  PROC DrawPart35()
    MoveL Offs(pOrigin,247.24,263.83,0.00),v40,z0,tPen\WObj:=wPaper;
    MoveL Offs(pOrigin,247.24,263.83,0.00),v40,z0,tPen\WObj:=wPaper;
    MoveL Offs(pOrigin,248.23,263.61,0.00),v40,z0,tPen\WObj:=wPaper;
    MoveL Offs(pOrigin,249.43,261.91,0.00),v40,z0,tPen\WObj:=wPaper;
    MoveL Offs(pOrigin,249.57,260.64,0.00),v40,z0,tPen\WObj:=wPaper;
    MoveL Offs(pOrigin,249.57,260.64,0.00),v40,z0,tPen\WObj:=wPaper;
    MoveL Offs(pOrigin,250.00,259.58,0.00),v40,z0,tPen\WObj:=wPaper;
    MoveL Offs(pOrigin,249.57,260.64,0.00),v40,z0,tPen\WObj:=wPaper;
    MoveL Offs(pOrigin,248.58,260.85,0.00),v40,z0,tPen\WObj:=wPaper;
    MoveL Offs(pOrigin,248.09,262.34,0.00),v40,z0,tPen\WObj:=wPaper;
    MoveL Offs(pOrigin,248.09,262.34,0.00),v40,z0,tPen\WObj:=wPaper;
    MoveL Offs(pOrigin,247.45,262.76,0.00),v40,z0,tPen\WObj:=wPaper;
    MoveL Offs(pOrigin,247.24,263.83,0.00),v40,fine,tPen\WObj:=wPaper;
    MoveL Offs(pOrigin,247.24,263.83,6.00),v60,z5,tPen\WObj:=wPaper;
    MoveL Offs(pOrigin,249.15,263.83,6.00),vTravel,z5,tPen\WObj:=wPaper;
    MoveL Offs(pOrigin,249.15,263.83,0.00),v60,z0,tPen\WObj:=wPaper;
    MoveL Offs(pOrigin,248.94,264.46,0.00),v40,z0,tPen\WObj:=wPaper;
    MoveL Offs(pOrigin,249.36,265.31,0.00),v40,z0,tPen\WObj:=wPaper;
    MoveL Offs(pOrigin,249.36,265.31,0.00),v40,z0,tPen\WObj:=wPaper;
    MoveL Offs(pOrigin,250.85,265.95,0.00),v40,z0,tPen\WObj:=wPaper;
    MoveL Offs(pOrigin,252.76,268.29,0.00),v40,z0,tPen\WObj:=wPaper;
    MoveL Offs(pOrigin,254.25,269.28,0.00),v40,z0,tPen\WObj:=wPaper;
    MoveL Offs(pOrigin,257.23,269.99,0.00),v40,z0,tPen\WObj:=wPaper;
    MoveL Offs(pOrigin,262.11,269.99,0.00),v40,z0,tPen\WObj:=wPaper;
    MoveL Offs(pOrigin,264.88,269.35,0.00),v40,z0,tPen\WObj:=wPaper;
    MoveL Offs(pOrigin,267.00,268.36,0.00),v40,z0,tPen\WObj:=wPaper;
    MoveL Offs(pOrigin,267.85,267.23,0.00),v40,z0,tPen\WObj:=wPaper;
    MoveL Offs(pOrigin,267.85,266.80,0.00),v40,z0,tPen\WObj:=wPaper;
    MoveL Offs(pOrigin,268.06,267.15,0.00),v40,z0,tPen\WObj:=wPaper;
    MoveL Offs(pOrigin,268.91,267.23,0.00),v40,z0,tPen\WObj:=wPaper;
    MoveL Offs(pOrigin,270.40,266.59,0.00),v40,fine,tPen\WObj:=wPaper;
    MoveL Offs(pOrigin,270.40,266.59,6.00),v60,z5,tPen\WObj:=wPaper;
    MoveL Offs(pOrigin,272.74,265.95,6.00),vTravel,z5,tPen\WObj:=wPaper;
    MoveL Offs(pOrigin,272.74,265.95,0.00),v60,z0,tPen\WObj:=wPaper;
    MoveL Offs(pOrigin,269.76,265.74,0.00),v40,z0,tPen\WObj:=wPaper;
    MoveL Offs(pOrigin,267.85,266.80,0.00),v40,z0,tPen\WObj:=wPaper;
    MoveL Offs(pOrigin,267.85,266.80,0.00),v40,z0,tPen\WObj:=wPaper;
    MoveL Offs(pOrigin,266.36,266.80,0.00),v40,z0,tPen\WObj:=wPaper;
    MoveL Offs(pOrigin,265.51,267.51,0.00),v40,z0,tPen\WObj:=wPaper;
    MoveL Offs(pOrigin,262.96,268.29,0.00),v40,z0,tPen\WObj:=wPaper;
    MoveL Offs(pOrigin,261.05,267.44,0.00),v40,z0,tPen\WObj:=wPaper;
    MoveL Offs(pOrigin,261.05,267.44,0.00),v40,z0,tPen\WObj:=wPaper;
    MoveL Offs(pOrigin,260.20,268.43,0.00),v40,z0,tPen\WObj:=wPaper;
    MoveL Offs(pOrigin,258.29,268.50,0.00),v40,z0,tPen\WObj:=wPaper;
    MoveL Offs(pOrigin,257.44,267.79,0.00),v40,z0,tPen\WObj:=wPaper;
    MoveL Offs(pOrigin,255.74,267.51,0.00),v40,z0,tPen\WObj:=wPaper;
    MoveL Offs(pOrigin,253.82,266.16,0.00),v40,z0,tPen\WObj:=wPaper;
    MoveL Offs(pOrigin,253.61,265.52,0.00),v40,z0,tPen\WObj:=wPaper;
    MoveL Offs(pOrigin,253.61,265.52,0.00),v40,z0,tPen\WObj:=wPaper;
    MoveL Offs(pOrigin,253.82,264.67,0.00),v40,z0,tPen\WObj:=wPaper;
    MoveL Offs(pOrigin,253.40,264.25,0.00),v40,z0,tPen\WObj:=wPaper;
    MoveL Offs(pOrigin,252.76,264.25,0.00),v40,z0,tPen\WObj:=wPaper;
    MoveL Offs(pOrigin,252.55,265.10,0.00),v40,z0,tPen\WObj:=wPaper;
    MoveL Offs(pOrigin,252.98,265.52,0.00),v40,z0,tPen\WObj:=wPaper;
    MoveL Offs(pOrigin,253.61,265.52,0.00),v40,z0,tPen\WObj:=wPaper;
    MoveL Offs(pOrigin,253.82,264.46,0.00),v40,z0,tPen\WObj:=wPaper;
    MoveL Offs(pOrigin,255.31,264.67,0.00),v40,z0,tPen\WObj:=wPaper;
    MoveL Offs(pOrigin,258.08,264.46,0.00),v40,z0,tPen\WObj:=wPaper;
    MoveL Offs(pOrigin,259.14,265.67,0.00),v40,z0,tPen\WObj:=wPaper;
    MoveL Offs(pOrigin,260.77,266.23,0.00),v40,z0,tPen\WObj:=wPaper;
    MoveL Offs(pOrigin,261.05,267.44,0.00),v40,fine,tPen\WObj:=wPaper;
    MoveL Offs(pOrigin,261.05,267.44,6.00),v60,z5,tPen\WObj:=wPaper;
    MoveL Offs(pOrigin,259.56,265.95,6.00),vTravel,z5,tPen\WObj:=wPaper;
    MoveL Offs(pOrigin,259.56,265.95,0.00),v60,z0,tPen\WObj:=wPaper;
    MoveL Offs(pOrigin,257.44,267.51,0.00),v40,z0,tPen\WObj:=wPaper;
    MoveL Offs(pOrigin,257.23,266.80,0.00),v40,z0,tPen\WObj:=wPaper;
    MoveL Offs(pOrigin,257.51,266.02,0.00),v40,z0,tPen\WObj:=wPaper;
    MoveL Offs(pOrigin,258.92,265.74,0.00),v40,z0,tPen\WObj:=wPaper;
    MoveL Offs(pOrigin,258.71,265.31,0.00),v40,z0,tPen\WObj:=wPaper;
    MoveL Offs(pOrigin,258.92,265.74,0.00),v40,z0,tPen\WObj:=wPaper;
    MoveL Offs(pOrigin,258.71,265.31,0.00),v40,fine,tPen\WObj:=wPaper;
    MoveL Offs(pOrigin,258.71,265.31,6.00),v60,z5,tPen\WObj:=wPaper;
    MoveL Offs(pOrigin,257.65,261.27,6.00),vTravel,z5,tPen\WObj:=wPaper;
    MoveL Offs(pOrigin,257.65,261.27,0.00),v60,z0,tPen\WObj:=wPaper;
    MoveL Offs(pOrigin,254.04,262.12,0.00),v40,fine,tPen\WObj:=wPaper;
    MoveL Offs(pOrigin,254.04,262.12,6.00),v60,z5,tPen\WObj:=wPaper;
    MoveL Offs(pOrigin,253.40,260.85,6.00),vTravel,z5,tPen\WObj:=wPaper;
    MoveL Offs(pOrigin,253.40,260.85,0.00),v60,z0,tPen\WObj:=wPaper;
    MoveL Offs(pOrigin,253.82,260.64,0.00),v40,z0,tPen\WObj:=wPaper;
    MoveL Offs(pOrigin,253.40,260.85,0.00),v40,fine,tPen\WObj:=wPaper;
    MoveL Offs(pOrigin,253.40,260.85,6.00),v60,z5,tPen\WObj:=wPaper;
    MoveL Offs(pOrigin,254.68,260.21,6.00),vTravel,z5,tPen\WObj:=wPaper;
    MoveL Offs(pOrigin,254.68,260.21,0.00),v60,z0,tPen\WObj:=wPaper;
    MoveL Offs(pOrigin,255.10,260.00,0.00),v40,z0,tPen\WObj:=wPaper;
    MoveL Offs(pOrigin,254.68,260.21,0.00),v40,fine,tPen\WObj:=wPaper;
    MoveL Offs(pOrigin,254.68,260.21,6.00),v60,z5,tPen\WObj:=wPaper;
    MoveL Offs(pOrigin,251.91,261.49,6.00),vTravel,z5,tPen\WObj:=wPaper;
    MoveL Offs(pOrigin,251.91,261.49,0.00),v60,z0,tPen\WObj:=wPaper;
    MoveL Offs(pOrigin,255.31,259.72,0.00),v40,z0,tPen\WObj:=wPaper;
    MoveL Offs(pOrigin,259.99,258.51,0.00),v40,fine,tPen\WObj:=wPaper;
    MoveL Offs(pOrigin,259.99,258.51,6.00),v60,z5,tPen\WObj:=wPaper;
    MoveL Offs(pOrigin,263.39,265.10,6.00),vTravel,z5,tPen\WObj:=wPaper;
    MoveL Offs(pOrigin,263.39,265.10,0.00),v60,z0,tPen\WObj:=wPaper;
    MoveL Offs(pOrigin,264.88,265.81,0.00),v40,z0,tPen\WObj:=wPaper;
    MoveL Offs(pOrigin,265.94,266.80,0.00),v40,fine,tPen\WObj:=wPaper;
    MoveL Offs(pOrigin,265.94,266.80,6.00),v60,z5,tPen\WObj:=wPaper;
    MoveL Offs(pOrigin,252.55,265.10,6.00),vTravel,z5,tPen\WObj:=wPaper;
    MoveL Offs(pOrigin,252.55,265.10,0.00),v60,z0,tPen\WObj:=wPaper;
    MoveL Offs(pOrigin,252.55,265.31,0.00),v40,z0,tPen\WObj:=wPaper;
    MoveL Offs(pOrigin,251.70,264.25,0.00),v40,z0,tPen\WObj:=wPaper;
    MoveL Offs(pOrigin,251.27,264.25,0.00),v40,fine,tPen\WObj:=wPaper;
    MoveL Offs(pOrigin,251.27,264.25,6.00),v60,z5,tPen\WObj:=wPaper;
    MoveL Offs(pOrigin,249.15,264.46,6.00),vTravel,z5,tPen\WObj:=wPaper;
    MoveL Offs(pOrigin,249.15,264.46,0.00),v60,z0,tPen\WObj:=wPaper;
    MoveL Offs(pOrigin,249.36,264.89,0.00),v40,z0,tPen\WObj:=wPaper;
    MoveL Offs(pOrigin,249.15,264.46,0.00),v40,fine,tPen\WObj:=wPaper;
    MoveL Offs(pOrigin,249.15,264.46,6.00),v60,z5,tPen\WObj:=wPaper;
    MoveL Offs(pOrigin,249.15,265.74,6.00),vTravel,z5,tPen\WObj:=wPaper;
    MoveL Offs(pOrigin,249.15,265.74,0.00),v60,z0,tPen\WObj:=wPaper;
    MoveL Offs(pOrigin,250.43,266.59,0.00),v40,z0,tPen\WObj:=wPaper;
    MoveL Offs(pOrigin,251.06,266.59,0.00),v40,fine,tPen\WObj:=wPaper;
    MoveL Offs(pOrigin,251.06,266.59,6.00),v60,z5,tPen\WObj:=wPaper;
    MoveL Offs(pOrigin,249.15,265.74,6.00),vTravel,z5,tPen\WObj:=wPaper;
    MoveL Offs(pOrigin,249.15,265.74,0.00),v60,z0,tPen\WObj:=wPaper;
    MoveL Offs(pOrigin,248.73,265.95,0.00),v40,z0,tPen\WObj:=wPaper;
    MoveL Offs(pOrigin,248.73,266.59,0.00),v40,fine,tPen\WObj:=wPaper;
    MoveL Offs(pOrigin,248.73,266.59,6.00),v60,z5,tPen\WObj:=wPaper;
    MoveL Offs(pOrigin,246.60,270.41,6.00),vTravel,z5,tPen\WObj:=wPaper;
    MoveL Offs(pOrigin,246.60,270.41,0.00),v60,z0,tPen\WObj:=wPaper;
    MoveL Offs(pOrigin,247.02,270.84,0.00),v40,z0,tPen\WObj:=wPaper;
  ENDPROC

  PROC DrawPart36()
    MoveL Offs(pOrigin,246.60,270.41,0.00),v40,fine,tPen\WObj:=wPaper;
    MoveL Offs(pOrigin,246.60,270.41,6.00),v60,z5,tPen\WObj:=wPaper;
    MoveL Offs(pOrigin,245.54,269.77,6.00),vTravel,z5,tPen\WObj:=wPaper;
    MoveL Offs(pOrigin,245.54,269.77,0.00),v60,z0,tPen\WObj:=wPaper;
    MoveL Offs(pOrigin,244.69,270.41,0.00),v40,z0,tPen\WObj:=wPaper;
    MoveL Offs(pOrigin,243.34,272.33,0.00),v40,z0,tPen\WObj:=wPaper;
    MoveL Offs(pOrigin,242.35,276.58,0.00),v40,fine,tPen\WObj:=wPaper;
    MoveL Offs(pOrigin,242.35,276.58,6.00),v60,z5,tPen\WObj:=wPaper;
    MoveL Offs(pOrigin,247.24,273.17,6.00),vTravel,z5,tPen\WObj:=wPaper;
    MoveL Offs(pOrigin,247.24,273.17,0.00),v60,z0,tPen\WObj:=wPaper;
    MoveL Offs(pOrigin,247.45,273.60,0.00),v40,z0,tPen\WObj:=wPaper;
    MoveL Offs(pOrigin,247.24,273.17,0.00),v40,z0,tPen\WObj:=wPaper;
    MoveL Offs(pOrigin,247.02,272.54,0.00),v40,z0,tPen\WObj:=wPaper;
    MoveL Offs(pOrigin,247.38,273.81,0.00),v40,z0,tPen\WObj:=wPaper;
    MoveL Offs(pOrigin,248.30,275.09,0.00),v40,fine,tPen\WObj:=wPaper;
    MoveL Offs(pOrigin,248.30,275.09,6.00),v60,z5,tPen\WObj:=wPaper;
    MoveL Offs(pOrigin,249.36,261.70,6.00),vTravel,z5,tPen\WObj:=wPaper;
    MoveL Offs(pOrigin,249.36,261.70,0.00),v60,z0,tPen\WObj:=wPaper;
    MoveL Offs(pOrigin,249.15,262.12,0.00),v40,z0,tPen\WObj:=wPaper;
    MoveL Offs(pOrigin,249.36,261.70,0.00),v40,fine,tPen\WObj:=wPaper;
    MoveL Offs(pOrigin,249.36,261.70,6.00),v60,z5,tPen\WObj:=wPaper;
    MoveL Offs(pOrigin,248.30,261.06,6.00),vTravel,z5,tPen\WObj:=wPaper;
    MoveL Offs(pOrigin,248.30,261.06,0.00),v60,z0,tPen\WObj:=wPaper;
    MoveL Offs(pOrigin,248.09,261.49,0.00),v40,z0,tPen\WObj:=wPaper;
    MoveL Offs(pOrigin,248.30,261.06,0.00),v40,fine,tPen\WObj:=wPaper;
    MoveL Offs(pOrigin,248.30,261.06,6.00),v60,z5,tPen\WObj:=wPaper;
    MoveL Offs(pOrigin,247.24,259.79,6.00),vTravel,z5,tPen\WObj:=wPaper;
    MoveL Offs(pOrigin,247.24,259.79,0.00),v60,z0,tPen\WObj:=wPaper;
    MoveL Offs(pOrigin,247.02,260.21,0.00),v40,z0,tPen\WObj:=wPaper;
    MoveL Offs(pOrigin,247.24,259.79,0.00),v40,fine,tPen\WObj:=wPaper;
    MoveL Offs(pOrigin,247.24,259.79,6.00),v60,z5,tPen\WObj:=wPaper;
    MoveL Offs(pOrigin,204.74,265.52,6.00),vTravel,z5,tPen\WObj:=wPaper;
    MoveL Offs(pOrigin,204.74,265.52,0.00),v60,z0,tPen\WObj:=wPaper;
    MoveL Offs(pOrigin,203.89,265.31,0.00),v40,z0,tPen\WObj:=wPaper;
    MoveL Offs(pOrigin,203.25,265.95,0.00),v40,z0,tPen\WObj:=wPaper;
    MoveL Offs(pOrigin,203.25,265.95,0.00),v40,z0,tPen\WObj:=wPaper;
    MoveL Offs(pOrigin,202.19,267.23,0.00),v40,z0,tPen\WObj:=wPaper;
    MoveL Offs(pOrigin,202.19,267.23,0.00),v40,z0,tPen\WObj:=wPaper;
    MoveL Offs(pOrigin,202.40,268.29,0.00),v40,z0,tPen\WObj:=wPaper;
    MoveL Offs(pOrigin,202.19,268.71,0.00),v40,fine,tPen\WObj:=wPaper;
    MoveL Offs(pOrigin,202.19,268.71,6.00),v60,z5,tPen\WObj:=wPaper;
    MoveL Offs(pOrigin,202.19,267.23,6.00),vTravel,z5,tPen\WObj:=wPaper;
    MoveL Offs(pOrigin,202.19,267.23,0.00),v60,z0,tPen\WObj:=wPaper;
    MoveL Offs(pOrigin,201.34,266.80,0.00),v40,z0,tPen\WObj:=wPaper;
    MoveL Offs(pOrigin,200.91,266.02,0.00),v40,z0,tPen\WObj:=wPaper;
    MoveL Offs(pOrigin,203.25,265.95,0.00),v40,z0,tPen\WObj:=wPaper;
    MoveL Offs(pOrigin,203.68,265.31,0.00),v40,z0,tPen\WObj:=wPaper;
    MoveL Offs(pOrigin,202.82,263.83,0.00),v40,z0,tPen\WObj:=wPaper;
    MoveL Offs(pOrigin,202.82,263.83,0.00),v40,z0,tPen\WObj:=wPaper;
    MoveL Offs(pOrigin,203.11,261.27,0.00),v40,z0,tPen\WObj:=wPaper;
    MoveL Offs(pOrigin,204.10,260.21,0.00),v40,fine,tPen\WObj:=wPaper;
    MoveL Offs(pOrigin,204.10,260.21,6.00),v60,z5,tPen\WObj:=wPaper;
    MoveL Offs(pOrigin,202.82,263.83,6.00),vTravel,z5,tPen\WObj:=wPaper;
    MoveL Offs(pOrigin,202.82,263.83,0.00),v60,z0,tPen\WObj:=wPaper;
    MoveL Offs(pOrigin,200.27,264.46,0.00),v40,fine,tPen\WObj:=wPaper;
    MoveL Offs(pOrigin,200.27,264.46,6.00),v60,z5,tPen\WObj:=wPaper;
    MoveL Offs(pOrigin,199.85,267.65,6.00),vTravel,z5,tPen\WObj:=wPaper;
    MoveL Offs(pOrigin,199.85,267.65,0.00),v60,z0,tPen\WObj:=wPaper;
    MoveL Offs(pOrigin,199.43,267.86,0.00),v40,z0,tPen\WObj:=wPaper;
    MoveL Offs(pOrigin,199.43,268.50,0.00),v40,z0,tPen\WObj:=wPaper;
    MoveL Offs(pOrigin,199.43,268.50,0.00),v40,z0,tPen\WObj:=wPaper;
    MoveL Offs(pOrigin,200.84,270.20,0.00),v40,z0,tPen\WObj:=wPaper;
    MoveL Offs(pOrigin,200.49,271.26,0.00),v40,z0,tPen\WObj:=wPaper;
    MoveL Offs(pOrigin,200.49,271.26,0.00),v40,z0,tPen\WObj:=wPaper;
    MoveL Offs(pOrigin,201.55,274.45,0.00),v40,z0,tPen\WObj:=wPaper;
    MoveL Offs(pOrigin,201.34,275.09,0.00),v40,z0,tPen\WObj:=wPaper;
    MoveL Offs(pOrigin,201.34,275.09,0.00),v40,z0,tPen\WObj:=wPaper;
    MoveL Offs(pOrigin,202.90,278.27,0.00),v40,z0,tPen\WObj:=wPaper;
    MoveL Offs(pOrigin,203.25,279.76,0.00),v40,z0,tPen\WObj:=wPaper;
    MoveL Offs(pOrigin,203.25,279.76,0.00),v40,z0,tPen\WObj:=wPaper;
    MoveL Offs(pOrigin,204.17,280.61,0.00),v40,z0,tPen\WObj:=wPaper;
    MoveL Offs(pOrigin,204.95,282.74,0.00),v40,fine,tPen\WObj:=wPaper;
    MoveL Offs(pOrigin,204.95,282.74,6.00),v60,z5,tPen\WObj:=wPaper;
    MoveL Offs(pOrigin,204.95,284.44,6.00),vTravel,z5,tPen\WObj:=wPaper;
    MoveL Offs(pOrigin,204.95,284.44,0.00),v60,z0,tPen\WObj:=wPaper;
    MoveL Offs(pOrigin,204.31,283.66,0.00),v40,z0,tPen\WObj:=wPaper;
    MoveL Offs(pOrigin,203.46,283.66,0.00),v40,z0,tPen\WObj:=wPaper;
    MoveL Offs(pOrigin,203.25,285.08,0.00),v40,z0,tPen\WObj:=wPaper;
    MoveL Offs(pOrigin,203.25,285.08,0.00),v40,z0,tPen\WObj:=wPaper;
    MoveL Offs(pOrigin,204.45,285.71,0.00),v40,z0,tPen\WObj:=wPaper;
    MoveL Offs(pOrigin,206.23,289.54,0.00),v40,fine,tPen\WObj:=wPaper;
    MoveL Offs(pOrigin,206.23,289.54,6.00),v60,z5,tPen\WObj:=wPaper;
    MoveL Offs(pOrigin,204.95,290.17,6.00),vTravel,z5,tPen\WObj:=wPaper;
    MoveL Offs(pOrigin,204.95,290.17,0.00),v60,z0,tPen\WObj:=wPaper;
    MoveL Offs(pOrigin,205.45,290.39,0.00),v40,z0,tPen\WObj:=wPaper;
    MoveL Offs(pOrigin,206.86,292.73,0.00),v40,fine,tPen\WObj:=wPaper;
    MoveL Offs(pOrigin,206.86,292.73,6.00),v60,z5,tPen\WObj:=wPaper;
    MoveL Offs(pOrigin,204.52,291.02,6.00),vTravel,z5,tPen\WObj:=wPaper;
    MoveL Offs(pOrigin,204.52,291.02,0.00),v60,z0,tPen\WObj:=wPaper;
    MoveL Offs(pOrigin,204.74,291.45,0.00),v40,z0,tPen\WObj:=wPaper;
    MoveL Offs(pOrigin,204.52,291.02,0.00),v40,z0,tPen\WObj:=wPaper;
    MoveL Offs(pOrigin,204.52,290.39,0.00),v40,z0,tPen\WObj:=wPaper;
    MoveL Offs(pOrigin,204.31,290.81,0.00),v40,z0,tPen\WObj:=wPaper;
    MoveL Offs(pOrigin,204.74,291.66,0.00),v40,z0,tPen\WObj:=wPaper;
    MoveL Offs(pOrigin,208.14,295.70,0.00),v40,fine,tPen\WObj:=wPaper;
    MoveL Offs(pOrigin,208.14,295.70,6.00),v60,z5,tPen\WObj:=wPaper;
    MoveL Offs(pOrigin,205.80,296.55,6.00),vTravel,z5,tPen\WObj:=wPaper;
    MoveL Offs(pOrigin,205.80,296.55,0.00),v60,z0,tPen\WObj:=wPaper;
    MoveL Offs(pOrigin,204.95,294.85,0.00),v40,z0,tPen\WObj:=wPaper;
    MoveL Offs(pOrigin,201.48,290.81,0.00),v40,z0,tPen\WObj:=wPaper;
    MoveL Offs(pOrigin,198.57,285.50,0.00),v40,z0,tPen\WObj:=wPaper;
    MoveL Offs(pOrigin,198.57,285.50,0.00),v40,z0,tPen\WObj:=wPaper;
    MoveL Offs(pOrigin,198.50,284.44,0.00),v40,z0,tPen\WObj:=wPaper;
    MoveL Offs(pOrigin,196.95,282.52,0.00),v40,z0,tPen\WObj:=wPaper;
    MoveL Offs(pOrigin,196.66,281.67,0.00),v40,z0,tPen\WObj:=wPaper;
    MoveL Offs(pOrigin,196.88,281.11,0.00),v40,z0,tPen\WObj:=wPaper;
    MoveL Offs(pOrigin,197.30,281.04,0.00),v40,z0,tPen\WObj:=wPaper;
    MoveL Offs(pOrigin,197.30,281.04,0.00),v40,z0,tPen\WObj:=wPaper;
    MoveL Offs(pOrigin,198.57,281.89,0.00),v40,z0,tPen\WObj:=wPaper;
    MoveL Offs(pOrigin,201.98,286.35,0.00),v40,z0,tPen\WObj:=wPaper;
    MoveL Offs(pOrigin,201.98,286.35,0.00),v40,z0,tPen\WObj:=wPaper;
    MoveL Offs(pOrigin,203.11,287.84,0.00),v40,z0,tPen\WObj:=wPaper;
    MoveL Offs(pOrigin,203.68,289.75,0.00),v40,z0,tPen\WObj:=wPaper;
    MoveL Offs(pOrigin,203.68,289.75,0.00),v40,z0,tPen\WObj:=wPaper;
    MoveL Offs(pOrigin,203.04,290.60,0.00),v40,z0,tPen\WObj:=wPaper;
    MoveL Offs(pOrigin,203.25,291.88,0.00),v40,z0,tPen\WObj:=wPaper;
    MoveL Offs(pOrigin,203.04,292.30,0.00),v40,z0,tPen\WObj:=wPaper;
    MoveL Offs(pOrigin,203.46,292.94,0.00),v40,z0,tPen\WObj:=wPaper;
    MoveL Offs(pOrigin,203.89,293.36,0.00),v40,z0,tPen\WObj:=wPaper;
    MoveL Offs(pOrigin,203.46,292.94,0.00),v40,fine,tPen\WObj:=wPaper;
  ENDPROC

  PROC DrawPart37()
    MoveL Offs(pOrigin,203.46,292.94,6.00),v60,z5,tPen\WObj:=wPaper;
    MoveL Offs(pOrigin,200.49,292.94,6.00),vTravel,z5,tPen\WObj:=wPaper;
    MoveL Offs(pOrigin,200.49,292.94,0.00),v60,z0,tPen\WObj:=wPaper;
    MoveL Offs(pOrigin,203.46,296.76,0.00),v40,z0,tPen\WObj:=wPaper;
    MoveL Offs(pOrigin,203.46,296.76,0.00),v40,z0,tPen\WObj:=wPaper;
    MoveL Offs(pOrigin,205.59,297.19,0.00),v40,z0,tPen\WObj:=wPaper;
    MoveL Offs(pOrigin,205.59,297.19,0.00),v40,z0,tPen\WObj:=wPaper;
    MoveL Offs(pOrigin,206.44,298.89,0.00),v40,fine,tPen\WObj:=wPaper;
    MoveL Offs(pOrigin,206.44,298.89,6.00),v60,z5,tPen\WObj:=wPaper;
    MoveL Offs(pOrigin,206.01,300.16,6.00),vTravel,z5,tPen\WObj:=wPaper;
    MoveL Offs(pOrigin,206.01,300.16,0.00),v60,z0,tPen\WObj:=wPaper;
    MoveL Offs(pOrigin,205.80,299.95,0.00),v40,z0,tPen\WObj:=wPaper;
    MoveL Offs(pOrigin,205.59,300.16,0.00),v40,z0,tPen\WObj:=wPaper;
    MoveL Offs(pOrigin,206.01,300.38,0.00),v40,z0,tPen\WObj:=wPaper;
    MoveL Offs(pOrigin,206.01,300.38,0.00),v40,z0,tPen\WObj:=wPaper;
    MoveL Offs(pOrigin,206.23,301.44,0.00),v40,z0,tPen\WObj:=wPaper;
    MoveL Offs(pOrigin,206.23,301.44,0.00),v40,z0,tPen\WObj:=wPaper;
    MoveL Offs(pOrigin,207.29,301.86,0.00),v40,z0,tPen\WObj:=wPaper;
    MoveL Offs(pOrigin,207.29,301.86,0.00),v40,z0,tPen\WObj:=wPaper;
    MoveL Offs(pOrigin,207.71,304.62,0.00),v40,z0,tPen\WObj:=wPaper;
    MoveL Offs(pOrigin,207.71,304.62,0.00),v40,z0,tPen\WObj:=wPaper;
    MoveL Offs(pOrigin,206.01,304.48,0.00),v40,z0,tPen\WObj:=wPaper;
    MoveL Offs(pOrigin,205.16,305.05,0.00),v40,z0,tPen\WObj:=wPaper;
    MoveL Offs(pOrigin,204.10,305.05,0.00),v40,z0,tPen\WObj:=wPaper;
    MoveL Offs(pOrigin,201.55,304.27,0.00),v40,z0,tPen\WObj:=wPaper;
    MoveL Offs(pOrigin,197.94,302.22,0.00),v40,z0,tPen\WObj:=wPaper;
    MoveL Offs(pOrigin,196.88,301.23,0.00),v40,z0,tPen\WObj:=wPaper;
    MoveL Offs(pOrigin,195.32,298.89,0.00),v40,z0,tPen\WObj:=wPaper;
    MoveL Offs(pOrigin,194.25,295.91,0.00),v40,z0,tPen\WObj:=wPaper;
    MoveL Offs(pOrigin,193.26,295.06,0.00),v40,z0,tPen\WObj:=wPaper;
    MoveL Offs(pOrigin,193.26,295.06,0.00),v40,z0,tPen\WObj:=wPaper;
    MoveL Offs(pOrigin,192.77,292.30,0.00),v40,z0,tPen\WObj:=wPaper;
    MoveL Offs(pOrigin,193.90,291.45,0.00),v40,z0,tPen\WObj:=wPaper;
    MoveL Offs(pOrigin,193.90,291.45,0.00),v40,z0,tPen\WObj:=wPaper;
    MoveL Offs(pOrigin,192.62,290.60,0.00),v40,z0,tPen\WObj:=wPaper;
    MoveL Offs(pOrigin,192.41,291.02,0.00),v40,z0,tPen\WObj:=wPaper;
    MoveL Offs(pOrigin,192.41,291.02,0.00),v40,z0,tPen\WObj:=wPaper;
    MoveL Offs(pOrigin,192.62,292.09,0.00),v40,z0,tPen\WObj:=wPaper;
    MoveL Offs(pOrigin,192.41,291.02,0.00),v40,z0,tPen\WObj:=wPaper;
    MoveL Offs(pOrigin,191.35,291.52,0.00),v40,z0,tPen\WObj:=wPaper;
    MoveL Offs(pOrigin,190.85,292.51,0.00),v40,z0,tPen\WObj:=wPaper;
    MoveL Offs(pOrigin,189.86,295.91,0.00),v40,z0,tPen\WObj:=wPaper;
    MoveL Offs(pOrigin,189.65,298.04,0.00),v40,z0,tPen\WObj:=wPaper;
    MoveL Offs(pOrigin,190.43,301.23,0.00),v40,z0,tPen\WObj:=wPaper;
    MoveL Offs(pOrigin,192.70,305.48,0.00),v40,z0,tPen\WObj:=wPaper;
    MoveL Offs(pOrigin,193.48,307.60,0.00),v40,z0,tPen\WObj:=wPaper;
    MoveL Offs(pOrigin,193.48,307.60,0.00),v40,z0,tPen\WObj:=wPaper;
    MoveL Offs(pOrigin,194.75,307.95,0.00),v40,z0,tPen\WObj:=wPaper;
    MoveL Offs(pOrigin,195.81,309.09,0.00),v40,z0,tPen\WObj:=wPaper;
    MoveL Offs(pOrigin,195.81,309.09,0.00),v40,z0,tPen\WObj:=wPaper;
    MoveL Offs(pOrigin,196.45,310.15,0.00),v40,z0,tPen\WObj:=wPaper;
    MoveL Offs(pOrigin,199.00,311.50,0.00),v40,z0,tPen\WObj:=wPaper;
    MoveL Offs(pOrigin,201.12,312.06,0.00),v40,z0,tPen\WObj:=wPaper;
    MoveL Offs(pOrigin,203.46,312.06,0.00),v40,z0,tPen\WObj:=wPaper;
    MoveL Offs(pOrigin,207.71,310.43,0.00),v40,z0,tPen\WObj:=wPaper;
    MoveL Offs(pOrigin,209.62,309.09,0.00),v40,z0,tPen\WObj:=wPaper;
    MoveL Offs(pOrigin,210.26,308.02,0.00),v40,z0,tPen\WObj:=wPaper;
    MoveL Offs(pOrigin,210.26,308.02,0.00),v40,z0,tPen\WObj:=wPaper;
    MoveL Offs(pOrigin,212.39,307.60,0.00),v40,z0,tPen\WObj:=wPaper;
    MoveL Offs(pOrigin,214.73,307.81,0.00),v40,z0,tPen\WObj:=wPaper;
    MoveL Offs(pOrigin,218.34,307.60,0.00),v40,fine,tPen\WObj:=wPaper;
    MoveL Offs(pOrigin,218.34,307.60,6.00),v60,z5,tPen\WObj:=wPaper;
    MoveL Offs(pOrigin,215.79,306.33,6.00),vTravel,z5,tPen\WObj:=wPaper;
    MoveL Offs(pOrigin,215.79,306.33,0.00),v60,z0,tPen\WObj:=wPaper;
    MoveL Offs(pOrigin,210.69,306.11,0.00),v40,z0,tPen\WObj:=wPaper;
    MoveL Offs(pOrigin,209.77,306.96,0.00),v40,z0,tPen\WObj:=wPaper;
    MoveL Offs(pOrigin,210.26,308.02,0.00),v40,fine,tPen\WObj:=wPaper;
    MoveL Offs(pOrigin,210.26,308.02,6.00),v60,z5,tPen\WObj:=wPaper;
    MoveL Offs(pOrigin,207.93,307.39,6.00),vTravel,z5,tPen\WObj:=wPaper;
    MoveL Offs(pOrigin,207.93,307.39,0.00),v60,z0,tPen\WObj:=wPaper;
    MoveL Offs(pOrigin,207.93,307.81,0.00),v40,z0,tPen\WObj:=wPaper;
    MoveL Offs(pOrigin,206.86,308.66,0.00),v40,fine,tPen\WObj:=wPaper;
    MoveL Offs(pOrigin,206.86,308.66,6.00),v60,z5,tPen\WObj:=wPaper;
    MoveL Offs(pOrigin,203.89,308.02,6.00),vTravel,z5,tPen\WObj:=wPaper;
    MoveL Offs(pOrigin,203.89,308.02,0.00),v60,z0,tPen\WObj:=wPaper;
    MoveL Offs(pOrigin,203.89,306.96,0.00),v40,fine,tPen\WObj:=wPaper;
    MoveL Offs(pOrigin,203.89,306.96,6.00),v60,z5,tPen\WObj:=wPaper;
    MoveL Offs(pOrigin,200.91,305.90,6.00),vTravel,z5,tPen\WObj:=wPaper;
    MoveL Offs(pOrigin,200.91,305.90,0.00),v60,z0,tPen\WObj:=wPaper;
    MoveL Offs(pOrigin,204.31,306.96,0.00),v40,z0,tPen\WObj:=wPaper;
    MoveL Offs(pOrigin,207.29,306.96,0.00),v40,z0,tPen\WObj:=wPaper;
    MoveL Offs(pOrigin,208.35,307.39,0.00),v40,z0,tPen\WObj:=wPaper;
    MoveL Offs(pOrigin,209.20,307.32,0.00),v40,z0,tPen\WObj:=wPaper;
    MoveL Offs(pOrigin,209.34,306.75,0.00),v40,z0,tPen\WObj:=wPaper;
    MoveL Offs(pOrigin,208.14,304.62,0.00),v40,z0,tPen\WObj:=wPaper;
    MoveL Offs(pOrigin,208.14,304.62,0.00),v40,z0,tPen\WObj:=wPaper;
    MoveL Offs(pOrigin,209.41,304.20,0.00),v40,z0,tPen\WObj:=wPaper;
    MoveL Offs(pOrigin,214.73,305.05,0.00),v40,fine,tPen\WObj:=wPaper;
    MoveL Offs(pOrigin,214.73,305.05,6.00),v60,z5,tPen\WObj:=wPaper;
    MoveL Offs(pOrigin,213.45,303.56,6.00),vTravel,z5,tPen\WObj:=wPaper;
    MoveL Offs(pOrigin,213.45,303.56,0.00),v60,z0,tPen\WObj:=wPaper;
    MoveL Offs(pOrigin,207.71,301.65,0.00),v40,z0,tPen\WObj:=wPaper;
    MoveL Offs(pOrigin,207.29,301.86,0.00),v40,z0,tPen\WObj:=wPaper;
    MoveL Offs(pOrigin,206.23,301.44,0.00),v40,z0,tPen\WObj:=wPaper;
    MoveL Offs(pOrigin,205.59,301.86,0.00),v40,z0,tPen\WObj:=wPaper;
    MoveL Offs(pOrigin,203.68,301.51,0.00),v40,z0,tPen\WObj:=wPaper;
    MoveL Offs(pOrigin,199.21,298.89,0.00),v40,z0,tPen\WObj:=wPaper;
    MoveL Offs(pOrigin,197.30,296.98,0.00),v40,z0,tPen\WObj:=wPaper;
    MoveL Offs(pOrigin,193.90,291.45,0.00),v40,z0,tPen\WObj:=wPaper;
    MoveL Offs(pOrigin,193.69,291.02,0.00),v40,z0,tPen\WObj:=wPaper;
    MoveL Offs(pOrigin,193.90,291.45,0.00),v40,z0,tPen\WObj:=wPaper;
    MoveL Offs(pOrigin,193.69,291.02,0.00),v40,fine,tPen\WObj:=wPaper;
    MoveL Offs(pOrigin,193.69,291.02,6.00),v60,z5,tPen\WObj:=wPaper;
    MoveL Offs(pOrigin,192.41,290.60,6.00),vTravel,z5,tPen\WObj:=wPaper;
    MoveL Offs(pOrigin,192.41,290.60,0.00),v60,z0,tPen\WObj:=wPaper;
    MoveL Offs(pOrigin,191.77,288.48,0.00),v40,z0,tPen\WObj:=wPaper;
    MoveL Offs(pOrigin,191.77,286.35,0.00),v40,z0,tPen\WObj:=wPaper;
    MoveL Offs(pOrigin,191.77,286.35,0.00),v40,z0,tPen\WObj:=wPaper;
    MoveL Offs(pOrigin,191.56,284.44,0.00),v40,z0,tPen\WObj:=wPaper;
    MoveL Offs(pOrigin,191.77,282.52,0.00),v40,z0,tPen\WObj:=wPaper;
    MoveL Offs(pOrigin,192.20,281.67,0.00),v40,z0,tPen\WObj:=wPaper;
    MoveL Offs(pOrigin,193.05,281.25,0.00),v40,z0,tPen\WObj:=wPaper;
    MoveL Offs(pOrigin,193.05,281.25,0.00),v40,z0,tPen\WObj:=wPaper;
    MoveL Offs(pOrigin,193.69,281.89,0.00),v40,z0,tPen\WObj:=wPaper;
    MoveL Offs(pOrigin,194.32,283.59,0.00),v40,z0,tPen\WObj:=wPaper;
    MoveL Offs(pOrigin,194.32,283.59,0.00),v40,z0,tPen\WObj:=wPaper;
    MoveL Offs(pOrigin,195.60,283.87,0.00),v40,z0,tPen\WObj:=wPaper;
    MoveL Offs(pOrigin,198.57,285.50,0.00),v40,fine,tPen\WObj:=wPaper;
    MoveL Offs(pOrigin,198.57,285.50,6.00),v60,z5,tPen\WObj:=wPaper;
    MoveL Offs(pOrigin,199.85,287.41,6.00),vTravel,z5,tPen\WObj:=wPaper;
  ENDPROC

  PROC DrawPart38()
    MoveL Offs(pOrigin,199.85,287.41,0.00),v60,z0,tPen\WObj:=wPaper;
    MoveL Offs(pOrigin,200.06,287.84,0.00),v40,z0,tPen\WObj:=wPaper;
    MoveL Offs(pOrigin,199.85,287.41,0.00),v40,fine,tPen\WObj:=wPaper;
    MoveL Offs(pOrigin,199.85,287.41,6.00),v60,z5,tPen\WObj:=wPaper;
    MoveL Offs(pOrigin,201.98,286.35,6.00),vTravel,z5,tPen\WObj:=wPaper;
    MoveL Offs(pOrigin,201.98,286.35,0.00),v60,z0,tPen\WObj:=wPaper;
    MoveL Offs(pOrigin,202.61,285.71,0.00),v40,z0,tPen\WObj:=wPaper;
    MoveL Offs(pOrigin,203.04,285.71,0.00),v40,z0,tPen\WObj:=wPaper;
    MoveL Offs(pOrigin,203.04,285.71,0.00),v40,z0,tPen\WObj:=wPaper;
    MoveL Offs(pOrigin,203.25,286.56,0.00),v40,z0,tPen\WObj:=wPaper;
    MoveL Offs(pOrigin,202.82,286.99,0.00),v40,z0,tPen\WObj:=wPaper;
    MoveL Offs(pOrigin,203.04,287.41,0.00),v40,z0,tPen\WObj:=wPaper;
    MoveL Offs(pOrigin,203.25,287.84,0.00),v40,z0,tPen\WObj:=wPaper;
    MoveL Offs(pOrigin,203.04,287.41,0.00),v40,fine,tPen\WObj:=wPaper;
    MoveL Offs(pOrigin,203.04,287.41,6.00),v60,z5,tPen\WObj:=wPaper;
    MoveL Offs(pOrigin,202.19,285.92,6.00),vTravel,z5,tPen\WObj:=wPaper;
    MoveL Offs(pOrigin,202.19,285.92,0.00),v60,z0,tPen\WObj:=wPaper;
    MoveL Offs(pOrigin,201.98,286.35,0.00),v40,z0,tPen\WObj:=wPaper;
    MoveL Offs(pOrigin,202.19,285.92,0.00),v40,fine,tPen\WObj:=wPaper;
    MoveL Offs(pOrigin,202.19,285.92,6.00),v60,z5,tPen\WObj:=wPaper;
    MoveL Offs(pOrigin,203.25,283.59,6.00),vTravel,z5,tPen\WObj:=wPaper;
    MoveL Offs(pOrigin,203.25,283.59,0.00),v60,z0,tPen\WObj:=wPaper;
    MoveL Offs(pOrigin,201.98,282.31,0.00),v40,z0,tPen\WObj:=wPaper;
    MoveL Offs(pOrigin,199.35,278.27,0.00),v40,z0,tPen\WObj:=wPaper;
    MoveL Offs(pOrigin,196.66,275.73,0.00),v40,z0,tPen\WObj:=wPaper;
    MoveL Offs(pOrigin,196.66,275.73,0.00),v40,z0,tPen\WObj:=wPaper;
    MoveL Offs(pOrigin,196.66,274.02,0.00),v40,z0,tPen\WObj:=wPaper;
    MoveL Offs(pOrigin,197.09,273.60,0.00),v40,z0,tPen\WObj:=wPaper;
    MoveL Offs(pOrigin,197.94,274.24,0.00),v40,z0,tPen\WObj:=wPaper;
    MoveL Offs(pOrigin,198.36,275.09,0.00),v40,z0,tPen\WObj:=wPaper;
    MoveL Offs(pOrigin,198.01,276.58,0.00),v40,z0,tPen\WObj:=wPaper;
    MoveL Offs(pOrigin,197.51,276.36,0.00),v40,z0,tPen\WObj:=wPaper;
    MoveL Offs(pOrigin,197.51,277.00,0.00),v40,z0,tPen\WObj:=wPaper;
    MoveL Offs(pOrigin,195.60,277.21,0.00),v40,z0,tPen\WObj:=wPaper;
    MoveL Offs(pOrigin,194.75,277.85,0.00),v40,z0,tPen\WObj:=wPaper;
    MoveL Offs(pOrigin,194.75,277.85,0.00),v40,z0,tPen\WObj:=wPaper;
    MoveL Offs(pOrigin,195.39,278.70,0.00),v40,z0,tPen\WObj:=wPaper;
    MoveL Offs(pOrigin,196.88,279.34,0.00),v40,z0,tPen\WObj:=wPaper;
    MoveL Offs(pOrigin,197.30,281.04,0.00),v40,z0,tPen\WObj:=wPaper;
    MoveL Offs(pOrigin,196.66,281.04,0.00),v40,z0,tPen\WObj:=wPaper;
    MoveL Offs(pOrigin,195.81,280.83,0.00),v40,z0,tPen\WObj:=wPaper;
    MoveL Offs(pOrigin,195.39,280.19,0.00),v40,z0,tPen\WObj:=wPaper;
    MoveL Offs(pOrigin,195.39,280.19,0.00),v40,z0,tPen\WObj:=wPaper;
    MoveL Offs(pOrigin,195.39,278.91,0.00),v40,fine,tPen\WObj:=wPaper;
    MoveL Offs(pOrigin,195.39,278.91,6.00),v60,z5,tPen\WObj:=wPaper;
    MoveL Offs(pOrigin,194.75,277.85,6.00),vTravel,z5,tPen\WObj:=wPaper;
    MoveL Offs(pOrigin,194.75,277.85,0.00),v60,z0,tPen\WObj:=wPaper;
    MoveL Offs(pOrigin,194.32,277.64,0.00),v40,z0,tPen\WObj:=wPaper;
    MoveL Offs(pOrigin,194.32,277.00,0.00),v40,z0,tPen\WObj:=wPaper;
    MoveL Offs(pOrigin,194.96,275.73,0.00),v40,fine,tPen\WObj:=wPaper;
    MoveL Offs(pOrigin,194.96,275.73,6.00),v60,z5,tPen\WObj:=wPaper;
    MoveL Offs(pOrigin,196.66,275.73,6.00),vTravel,z5,tPen\WObj:=wPaper;
    MoveL Offs(pOrigin,196.66,275.73,0.00),v60,z0,tPen\WObj:=wPaper;
    MoveL Offs(pOrigin,195.39,275.73,0.00),v40,z0,tPen\WObj:=wPaper;
    MoveL Offs(pOrigin,194.96,275.30,0.00),v40,z0,tPen\WObj:=wPaper;
    MoveL Offs(pOrigin,195.39,274.24,0.00),v40,z0,tPen\WObj:=wPaper;
    MoveL Offs(pOrigin,196.45,273.74,0.00),v40,z0,tPen\WObj:=wPaper;
    MoveL Offs(pOrigin,196.88,271.48,0.00),v40,z0,tPen\WObj:=wPaper;
    MoveL Offs(pOrigin,197.94,271.05,0.00),v40,fine,tPen\WObj:=wPaper;
    MoveL Offs(pOrigin,197.94,271.05,6.00),v60,z5,tPen\WObj:=wPaper;
    MoveL Offs(pOrigin,199.00,269.35,6.00),vTravel,z5,tPen\WObj:=wPaper;
    MoveL Offs(pOrigin,199.00,269.35,0.00),v60,z0,tPen\WObj:=wPaper;
    MoveL Offs(pOrigin,198.22,269.77,0.00),v40,z0,tPen\WObj:=wPaper;
    MoveL Offs(pOrigin,197.94,270.62,0.00),v40,z0,tPen\WObj:=wPaper;
    MoveL Offs(pOrigin,198.57,273.17,0.00),v40,z0,tPen\WObj:=wPaper;
    MoveL Offs(pOrigin,198.57,273.17,0.00),v40,z0,tPen\WObj:=wPaper;
    MoveL Offs(pOrigin,199.43,273.60,0.00),v40,z0,tPen\WObj:=wPaper;
    MoveL Offs(pOrigin,200.27,274.80,0.00),v40,z0,tPen\WObj:=wPaper;
    MoveL Offs(pOrigin,201.34,275.09,0.00),v40,fine,tPen\WObj:=wPaper;
    MoveL Offs(pOrigin,201.34,275.09,6.00),v60,z5,tPen\WObj:=wPaper;
    MoveL Offs(pOrigin,203.89,273.81,6.00),vTravel,z5,tPen\WObj:=wPaper;
    MoveL Offs(pOrigin,203.89,273.81,0.00),v60,z0,tPen\WObj:=wPaper;
    MoveL Offs(pOrigin,203.68,275.30,0.00),v40,z0,tPen\WObj:=wPaper;
    MoveL Offs(pOrigin,205.38,279.55,0.00),v40,fine,tPen\WObj:=wPaper;
    MoveL Offs(pOrigin,205.38,279.55,6.00),v60,z5,tPen\WObj:=wPaper;
    MoveL Offs(pOrigin,203.25,279.76,6.00),vTravel,z5,tPen\WObj:=wPaper;
    MoveL Offs(pOrigin,203.25,279.76,0.00),v60,z0,tPen\WObj:=wPaper;
    MoveL Offs(pOrigin,203.04,280.19,0.00),v40,z0,tPen\WObj:=wPaper;
    MoveL Offs(pOrigin,203.25,282.10,0.00),v40,z0,tPen\WObj:=wPaper;
    MoveL Offs(pOrigin,202.82,282.74,0.00),v40,fine,tPen\WObj:=wPaper;
    MoveL Offs(pOrigin,202.82,282.74,6.00),v60,z5,tPen\WObj:=wPaper;
    MoveL Offs(pOrigin,205.16,287.20,6.00),vTravel,z5,tPen\WObj:=wPaper;
    MoveL Offs(pOrigin,205.16,287.20,0.00),v60,z0,tPen\WObj:=wPaper;
    MoveL Offs(pOrigin,205.38,287.62,0.00),v40,z0,tPen\WObj:=wPaper;
    MoveL Offs(pOrigin,205.16,287.20,0.00),v40,fine,tPen\WObj:=wPaper;
    MoveL Offs(pOrigin,205.16,287.20,6.00),v60,z5,tPen\WObj:=wPaper;
    MoveL Offs(pOrigin,199.64,291.66,6.00),vTravel,z5,tPen\WObj:=wPaper;
    MoveL Offs(pOrigin,199.64,291.66,0.00),v60,z0,tPen\WObj:=wPaper;
    MoveL Offs(pOrigin,199.64,291.45,0.00),v40,z0,tPen\WObj:=wPaper;
    MoveL Offs(pOrigin,200.27,291.88,0.00),v40,z0,tPen\WObj:=wPaper;
    MoveL Offs(pOrigin,200.49,292.94,0.00),v40,z0,tPen\WObj:=wPaper;
    MoveL Offs(pOrigin,200.49,292.94,0.00),v40,z0,tPen\WObj:=wPaper;
    MoveL Offs(pOrigin,200.06,292.94,0.00),v40,z0,tPen\WObj:=wPaper;
    MoveL Offs(pOrigin,199.21,292.09,0.00),v40,z0,tPen\WObj:=wPaper;
    MoveL Offs(pOrigin,199.64,291.66,0.00),v40,z0,tPen\WObj:=wPaper;
    MoveL Offs(pOrigin,199.21,291.45,0.00),v40,z0,tPen\WObj:=wPaper;
    MoveL Offs(pOrigin,196.80,287.41,0.00),v40,z0,tPen\WObj:=wPaper;
    MoveL Offs(pOrigin,195.60,284.01,0.00),v40,fine,tPen\WObj:=wPaper;
    MoveL Offs(pOrigin,195.60,284.01,6.00),v60,z5,tPen\WObj:=wPaper;
    MoveL Offs(pOrigin,194.32,283.59,6.00),vTravel,z5,tPen\WObj:=wPaper;
    MoveL Offs(pOrigin,194.32,283.59,0.00),v60,z0,tPen\WObj:=wPaper;
    MoveL Offs(pOrigin,194.11,284.86,0.00),v40,z0,tPen\WObj:=wPaper;
    MoveL Offs(pOrigin,194.75,287.41,0.00),v40,z0,tPen\WObj:=wPaper;
    MoveL Offs(pOrigin,194.32,287.84,0.00),v40,z0,tPen\WObj:=wPaper;
    MoveL Offs(pOrigin,194.32,287.84,0.00),v40,z0,tPen\WObj:=wPaper;
    MoveL Offs(pOrigin,197.94,293.79,0.00),v40,z0,tPen\WObj:=wPaper;
    MoveL Offs(pOrigin,200.70,296.55,0.00),v40,fine,tPen\WObj:=wPaper;
    MoveL Offs(pOrigin,200.70,296.55,6.00),v60,z5,tPen\WObj:=wPaper;
    MoveL Offs(pOrigin,199.64,295.49,6.00),vTravel,z5,tPen\WObj:=wPaper;
    MoveL Offs(pOrigin,199.64,295.49,0.00),v60,z0,tPen\WObj:=wPaper;
    MoveL Offs(pOrigin,200.06,295.91,0.00),v40,z0,tPen\WObj:=wPaper;
    MoveL Offs(pOrigin,199.64,295.49,0.00),v40,fine,tPen\WObj:=wPaper;
    MoveL Offs(pOrigin,199.64,295.49,6.00),v60,z5,tPen\WObj:=wPaper;
    MoveL Offs(pOrigin,196.02,294.85,6.00),vTravel,z5,tPen\WObj:=wPaper;
    MoveL Offs(pOrigin,196.02,294.85,0.00),v60,z0,tPen\WObj:=wPaper;
    MoveL Offs(pOrigin,196.45,295.49,0.00),v40,z0,tPen\WObj:=wPaper;
    MoveL Offs(pOrigin,196.02,294.85,0.00),v40,fine,tPen\WObj:=wPaper;
    MoveL Offs(pOrigin,196.02,294.85,6.00),v60,z5,tPen\WObj:=wPaper;
    MoveL Offs(pOrigin,193.26,295.06,6.00),vTravel,z5,tPen\WObj:=wPaper;
    MoveL Offs(pOrigin,193.26,295.06,0.00),v60,z0,tPen\WObj:=wPaper;
  ENDPROC

  PROC DrawPart39()
    MoveL Offs(pOrigin,192.70,295.49,0.00),v40,z0,tPen\WObj:=wPaper;
    MoveL Offs(pOrigin,192.41,296.76,0.00),v40,z0,tPen\WObj:=wPaper;
    MoveL Offs(pOrigin,192.41,299.52,0.00),v40,z0,tPen\WObj:=wPaper;
    MoveL Offs(pOrigin,192.41,299.52,0.00),v40,z0,tPen\WObj:=wPaper;
    MoveL Offs(pOrigin,193.55,300.16,0.00),v40,z0,tPen\WObj:=wPaper;
    MoveL Offs(pOrigin,194.96,302.92,0.00),v40,z0,tPen\WObj:=wPaper;
    MoveL Offs(pOrigin,195.18,304.20,0.00),v40,z0,tPen\WObj:=wPaper;
    MoveL Offs(pOrigin,195.18,304.20,0.00),v40,z0,tPen\WObj:=wPaper;
    MoveL Offs(pOrigin,199.00,307.03,0.00),v40,z0,tPen\WObj:=wPaper;
    MoveL Offs(pOrigin,201.34,307.81,0.00),v40,z0,tPen\WObj:=wPaper;
    MoveL Offs(pOrigin,203.04,307.81,0.00),v40,z0,tPen\WObj:=wPaper;
    MoveL Offs(pOrigin,204.95,308.66,0.00),v40,z0,tPen\WObj:=wPaper;
    MoveL Offs(pOrigin,206.79,308.88,0.00),v40,z0,tPen\WObj:=wPaper;
    MoveL Offs(pOrigin,206.79,309.30,0.00),v40,z0,tPen\WObj:=wPaper;
    MoveL Offs(pOrigin,206.01,309.80,0.00),v40,z0,tPen\WObj:=wPaper;
    MoveL Offs(pOrigin,203.68,310.36,0.00),v40,fine,tPen\WObj:=wPaper;
    MoveL Offs(pOrigin,203.68,310.36,6.00),v60,z5,tPen\WObj:=wPaper;
    MoveL Offs(pOrigin,205.80,304.41,6.00),vTravel,z5,tPen\WObj:=wPaper;
    MoveL Offs(pOrigin,205.80,304.41,0.00),v60,z0,tPen\WObj:=wPaper;
    MoveL Offs(pOrigin,205.38,303.85,0.00),v40,z0,tPen\WObj:=wPaper;
    MoveL Offs(pOrigin,200.91,302.08,0.00),v40,fine,tPen\WObj:=wPaper;
    MoveL Offs(pOrigin,200.91,302.08,6.00),v60,z5,tPen\WObj:=wPaper;
    MoveL Offs(pOrigin,196.88,301.01,6.00),vTravel,z5,tPen\WObj:=wPaper;
    MoveL Offs(pOrigin,196.88,301.01,0.00),v60,z0,tPen\WObj:=wPaper;
    MoveL Offs(pOrigin,197.73,301.86,0.00),v40,z0,tPen\WObj:=wPaper;
    MoveL Offs(pOrigin,196.88,301.01,0.00),v40,fine,tPen\WObj:=wPaper;
    MoveL Offs(pOrigin,196.88,301.01,6.00),v60,z5,tPen\WObj:=wPaper;
    MoveL Offs(pOrigin,194.54,302.71,6.00),vTravel,z5,tPen\WObj:=wPaper;
    MoveL Offs(pOrigin,194.54,302.71,0.00),v60,z0,tPen\WObj:=wPaper;
    MoveL Offs(pOrigin,193.69,303.35,0.00),v40,z0,tPen\WObj:=wPaper;
    MoveL Offs(pOrigin,194.32,303.99,0.00),v40,z0,tPen\WObj:=wPaper;
    MoveL Offs(pOrigin,195.18,304.20,0.00),v40,z0,tPen\WObj:=wPaper;
    MoveL Offs(pOrigin,195.18,304.20,0.00),v40,z0,tPen\WObj:=wPaper;
    MoveL Offs(pOrigin,196.02,304.84,0.00),v40,fine,tPen\WObj:=wPaper;
    MoveL Offs(pOrigin,196.02,304.84,6.00),v60,z5,tPen\WObj:=wPaper;
    MoveL Offs(pOrigin,193.69,303.14,6.00),vTravel,z5,tPen\WObj:=wPaper;
    MoveL Offs(pOrigin,193.69,303.14,0.00),v60,z0,tPen\WObj:=wPaper;
    MoveL Offs(pOrigin,192.84,302.29,0.00),v40,z0,tPen\WObj:=wPaper;
    MoveL Offs(pOrigin,192.41,302.29,0.00),v40,z0,tPen\WObj:=wPaper;
    MoveL Offs(pOrigin,192.41,302.29,0.00),v40,z0,tPen\WObj:=wPaper;
    MoveL Offs(pOrigin,191.77,303.35,0.00),v40,fine,tPen\WObj:=wPaper;
    MoveL Offs(pOrigin,191.77,303.35,6.00),v60,z5,tPen\WObj:=wPaper;
    MoveL Offs(pOrigin,192.41,302.29,6.00),vTravel,z5,tPen\WObj:=wPaper;
    MoveL Offs(pOrigin,192.41,302.29,0.00),v60,z0,tPen\WObj:=wPaper;
    MoveL Offs(pOrigin,192.20,300.80,0.00),v40,z0,tPen\WObj:=wPaper;
    MoveL Offs(pOrigin,192.41,299.52,0.00),v40,fine,tPen\WObj:=wPaper;
    MoveL Offs(pOrigin,192.41,299.52,6.00),v60,z5,tPen\WObj:=wPaper;
    MoveL Offs(pOrigin,195.18,298.25,6.00),vTravel,z5,tPen\WObj:=wPaper;
    MoveL Offs(pOrigin,195.18,298.25,0.00),v60,z0,tPen\WObj:=wPaper;
    MoveL Offs(pOrigin,195.39,298.67,0.00),v40,z0,tPen\WObj:=wPaper;
    MoveL Offs(pOrigin,195.18,298.25,0.00),v40,fine,tPen\WObj:=wPaper;
    MoveL Offs(pOrigin,195.18,298.25,6.00),v60,z5,tPen\WObj:=wPaper;
    MoveL Offs(pOrigin,203.46,296.76,6.00),vTravel,z5,tPen\WObj:=wPaper;
    MoveL Offs(pOrigin,203.46,296.76,0.00),v60,z0,tPen\WObj:=wPaper;
    MoveL Offs(pOrigin,202.82,297.19,0.00),v40,z0,tPen\WObj:=wPaper;
    MoveL Offs(pOrigin,201.12,296.55,0.00),v40,z0,tPen\WObj:=wPaper;
    MoveL Offs(pOrigin,200.84,296.98,0.00),v40,z0,tPen\WObj:=wPaper;
    MoveL Offs(pOrigin,201.12,297.61,0.00),v40,z0,tPen\WObj:=wPaper;
    MoveL Offs(pOrigin,204.74,300.23,0.00),v40,z0,tPen\WObj:=wPaper;
    MoveL Offs(pOrigin,205.59,300.38,0.00),v40,z0,tPen\WObj:=wPaper;
    MoveL Offs(pOrigin,206.01,300.38,0.00),v40,z0,tPen\WObj:=wPaper;
    MoveL Offs(pOrigin,206.44,299.95,0.00),v40,z0,tPen\WObj:=wPaper;
    MoveL Offs(pOrigin,206.51,299.10,0.00),v40,z0,tPen\WObj:=wPaper;
    MoveL Offs(pOrigin,206.86,299.03,0.00),v40,z0,tPen\WObj:=wPaper;
    MoveL Offs(pOrigin,211.32,301.23,0.00),v40,fine,tPen\WObj:=wPaper;
    MoveL Offs(pOrigin,211.32,301.23,6.00),v60,z5,tPen\WObj:=wPaper;
    MoveL Offs(pOrigin,209.84,298.46,6.00),vTravel,z5,tPen\WObj:=wPaper;
    MoveL Offs(pOrigin,209.84,298.46,0.00),v60,z0,tPen\WObj:=wPaper;
    MoveL Offs(pOrigin,207.29,296.62,0.00),v40,z0,tPen\WObj:=wPaper;
    MoveL Offs(pOrigin,206.44,296.34,0.00),v40,z0,tPen\WObj:=wPaper;
    MoveL Offs(pOrigin,205.80,296.55,0.00),v40,fine,tPen\WObj:=wPaper;
    MoveL Offs(pOrigin,205.80,296.55,6.00),v60,z5,tPen\WObj:=wPaper;
    MoveL Offs(pOrigin,214.09,307.81,6.00),vTravel,z5,tPen\WObj:=wPaper;
    MoveL Offs(pOrigin,214.09,307.81,0.00),v60,z0,tPen\WObj:=wPaper;
    MoveL Offs(pOrigin,213.88,309.30,0.00),v40,z0,tPen\WObj:=wPaper;
    MoveL Offs(pOrigin,213.88,309.30,0.00),v40,z0,tPen\WObj:=wPaper;
    MoveL Offs(pOrigin,216.21,309.51,0.00),v40,z0,tPen\WObj:=wPaper;
    MoveL Offs(pOrigin,216.21,309.51,0.00),v40,z0,tPen\WObj:=wPaper;
    MoveL Offs(pOrigin,214.94,311.07,0.00),v40,z0,tPen\WObj:=wPaper;
    MoveL Offs(pOrigin,214.09,311.00,0.00),v40,z0,tPen\WObj:=wPaper;
    MoveL Offs(pOrigin,213.02,311.50,0.00),v40,z0,tPen\WObj:=wPaper;
    MoveL Offs(pOrigin,210.90,314.19,0.00),v40,z0,tPen\WObj:=wPaper;
    MoveL Offs(pOrigin,210.48,314.40,0.00),v40,z0,tPen\WObj:=wPaper;
    MoveL Offs(pOrigin,208.35,315.75,0.00),v40,z0,tPen\WObj:=wPaper;
    MoveL Offs(pOrigin,204.74,316.95,0.00),v40,fine,tPen\WObj:=wPaper;
    MoveL Offs(pOrigin,204.74,316.95,6.00),v60,z5,tPen\WObj:=wPaper;
    MoveL Offs(pOrigin,200.27,317.59,6.00),vTravel,z5,tPen\WObj:=wPaper;
    MoveL Offs(pOrigin,200.27,317.59,0.00),v60,z0,tPen\WObj:=wPaper;
    MoveL Offs(pOrigin,200.70,318.01,0.00),v40,z0,tPen\WObj:=wPaper;
    MoveL Offs(pOrigin,200.27,317.59,0.00),v40,fine,tPen\WObj:=wPaper;
    MoveL Offs(pOrigin,200.27,317.59,6.00),v60,z5,tPen\WObj:=wPaper;
    MoveL Offs(pOrigin,199.85,316.31,6.00),vTravel,z5,tPen\WObj:=wPaper;
    MoveL Offs(pOrigin,199.85,316.31,0.00),v60,z0,tPen\WObj:=wPaper;
    MoveL Offs(pOrigin,198.79,315.46,0.00),v40,z0,tPen\WObj:=wPaper;
    MoveL Offs(pOrigin,198.79,314.83,0.00),v40,z0,tPen\WObj:=wPaper;
    MoveL Offs(pOrigin,198.79,314.83,0.00),v40,z0,tPen\WObj:=wPaper;
    MoveL Offs(pOrigin,199.43,314.26,0.00),v40,z0,tPen\WObj:=wPaper;
    MoveL Offs(pOrigin,203.68,314.83,0.00),v40,z0,tPen\WObj:=wPaper;
    MoveL Offs(pOrigin,206.44,314.05,0.00),v40,z0,tPen\WObj:=wPaper;
    MoveL Offs(pOrigin,211.96,310.08,0.00),v40,z0,tPen\WObj:=wPaper;
    MoveL Offs(pOrigin,213.88,309.30,0.00),v40,fine,tPen\WObj:=wPaper;
    MoveL Offs(pOrigin,213.88,309.30,6.00),v60,z5,tPen\WObj:=wPaper;
    MoveL Offs(pOrigin,214.51,311.21,6.00),vTravel,z5,tPen\WObj:=wPaper;
    MoveL Offs(pOrigin,214.51,311.21,0.00),v60,z0,tPen\WObj:=wPaper;
    MoveL Offs(pOrigin,214.09,313.34,0.00),v40,z0,tPen\WObj:=wPaper;
    MoveL Offs(pOrigin,214.09,313.34,0.00),v40,z0,tPen\WObj:=wPaper;
    MoveL Offs(pOrigin,212.81,317.80,0.00),v40,fine,tPen\WObj:=wPaper;
    MoveL Offs(pOrigin,212.81,317.80,6.00),v60,z5,tPen\WObj:=wPaper;
    MoveL Offs(pOrigin,212.60,319.71,6.00),vTravel,z5,tPen\WObj:=wPaper;
    MoveL Offs(pOrigin,212.60,319.71,0.00),v60,z0,tPen\WObj:=wPaper;
    MoveL Offs(pOrigin,212.81,318.23,0.00),v40,z0,tPen\WObj:=wPaper;
    MoveL Offs(pOrigin,212.39,317.87,0.00),v40,z0,tPen\WObj:=wPaper;
    MoveL Offs(pOrigin,209.20,320.00,0.00),v40,z0,tPen\WObj:=wPaper;
    MoveL Offs(pOrigin,205.59,320.56,0.00),v40,z0,tPen\WObj:=wPaper;
    MoveL Offs(pOrigin,202.61,319.43,0.00),v40,z0,tPen\WObj:=wPaper;
    MoveL Offs(pOrigin,200.70,318.23,0.00),v40,z0,tPen\WObj:=wPaper;
    MoveL Offs(pOrigin,199.99,317.38,0.00),v40,z0,tPen\WObj:=wPaper;
    MoveL Offs(pOrigin,199.85,316.31,0.00),v40,z0,tPen\WObj:=wPaper;
    MoveL Offs(pOrigin,199.85,316.31,0.00),v40,z0,tPen\WObj:=wPaper;
    MoveL Offs(pOrigin,204.31,316.95,0.00),v40,z0,tPen\WObj:=wPaper;
  ENDPROC

  PROC DrawPart40()
    MoveL Offs(pOrigin,205.16,317.66,0.00),v40,z0,tPen\WObj:=wPaper;
    MoveL Offs(pOrigin,206.23,317.80,0.00),v40,z0,tPen\WObj:=wPaper;
    MoveL Offs(pOrigin,209.84,316.81,0.00),v40,z0,tPen\WObj:=wPaper;
    MoveL Offs(pOrigin,211.75,315.67,0.00),v40,fine,tPen\WObj:=wPaper;
    MoveL Offs(pOrigin,211.75,315.67,6.00),v60,z5,tPen\WObj:=wPaper;
    MoveL Offs(pOrigin,212.18,312.49,6.00),vTravel,z5,tPen\WObj:=wPaper;
    MoveL Offs(pOrigin,212.18,312.49,0.00),v60,z0,tPen\WObj:=wPaper;
    MoveL Offs(pOrigin,211.96,312.91,0.00),v40,z0,tPen\WObj:=wPaper;
    MoveL Offs(pOrigin,212.18,312.49,0.00),v40,fine,tPen\WObj:=wPaper;
    MoveL Offs(pOrigin,212.18,312.49,6.00),v60,z5,tPen\WObj:=wPaper;
    MoveL Offs(pOrigin,214.09,313.34,6.00),vTravel,z5,tPen\WObj:=wPaper;
    MoveL Offs(pOrigin,214.09,313.34,0.00),v60,z0,tPen\WObj:=wPaper;
    MoveL Offs(pOrigin,215.36,312.91,0.00),v40,z0,tPen\WObj:=wPaper;
    MoveL Offs(pOrigin,217.27,311.07,0.00),v40,z0,tPen\WObj:=wPaper;
    MoveL Offs(pOrigin,218.12,310.79,0.00),v40,z0,tPen\WObj:=wPaper;
    MoveL Offs(pOrigin,218.76,311.00,0.00),v40,z0,tPen\WObj:=wPaper;
    MoveL Offs(pOrigin,218.76,311.00,0.00),v40,z0,tPen\WObj:=wPaper;
    MoveL Offs(pOrigin,218.34,312.91,0.00),v40,z0,tPen\WObj:=wPaper;
    MoveL Offs(pOrigin,218.34,312.91,0.00),v40,z0,tPen\WObj:=wPaper;
    MoveL Offs(pOrigin,218.34,314.40,0.00),v40,z0,tPen\WObj:=wPaper;
    MoveL Offs(pOrigin,218.34,314.40,0.00),v40,z0,tPen\WObj:=wPaper;
    MoveL Offs(pOrigin,217.35,315.11,0.00),v40,z0,tPen\WObj:=wPaper;
    MoveL Offs(pOrigin,216.85,316.95,0.00),v40,z0,tPen\WObj:=wPaper;
    MoveL Offs(pOrigin,217.27,320.14,0.00),v40,fine,tPen\WObj:=wPaper;
    MoveL Offs(pOrigin,217.27,320.14,6.00),v60,z5,tPen\WObj:=wPaper;
    MoveL Offs(pOrigin,218.76,316.95,6.00),vTravel,z5,tPen\WObj:=wPaper;
    MoveL Offs(pOrigin,218.76,316.95,0.00),v60,z0,tPen\WObj:=wPaper;
    MoveL Offs(pOrigin,218.34,317.38,0.00),v40,z0,tPen\WObj:=wPaper;
    MoveL Offs(pOrigin,218.34,318.65,0.00),v40,z0,tPen\WObj:=wPaper;
    MoveL Offs(pOrigin,218.98,320.99,0.00),v40,z0,tPen\WObj:=wPaper;
    MoveL Offs(pOrigin,218.98,323.54,0.00),v40,z0,tPen\WObj:=wPaper;
    MoveL Offs(pOrigin,218.69,324.81,0.00),v40,z0,tPen\WObj:=wPaper;
    MoveL Offs(pOrigin,217.91,325.88,0.00),v40,z0,tPen\WObj:=wPaper;
    MoveL Offs(pOrigin,217.06,326.30,0.00),v40,z0,tPen\WObj:=wPaper;
    MoveL Offs(pOrigin,217.35,326.16,0.00),v40,z0,tPen\WObj:=wPaper;
    MoveL Offs(pOrigin,214.51,327.43,0.00),v40,z0,tPen\WObj:=wPaper;
    MoveL Offs(pOrigin,213.88,328.21,0.00),v40,fine,tPen\WObj:=wPaper;
    MoveL Offs(pOrigin,213.88,328.21,6.00),v60,z5,tPen\WObj:=wPaper;
    MoveL Offs(pOrigin,214.94,325.24,6.00),vTravel,z5,tPen\WObj:=wPaper;
    MoveL Offs(pOrigin,214.94,325.24,0.00),v60,z0,tPen\WObj:=wPaper;
    MoveL Offs(pOrigin,213.02,326.09,0.00),v40,z0,tPen\WObj:=wPaper;
    MoveL Offs(pOrigin,209.62,326.09,0.00),v40,z0,tPen\WObj:=wPaper;
    MoveL Offs(pOrigin,208.99,326.51,0.00),v40,z0,tPen\WObj:=wPaper;
    MoveL Offs(pOrigin,208.99,326.51,0.00),v40,z0,tPen\WObj:=wPaper;
    MoveL Offs(pOrigin,209.62,327.43,0.00),v40,z0,tPen\WObj:=wPaper;
    MoveL Offs(pOrigin,213.24,328.00,0.00),v40,z0,tPen\WObj:=wPaper;
    MoveL Offs(pOrigin,214.51,328.64,0.00),v40,z0,tPen\WObj:=wPaper;
    MoveL Offs(pOrigin,217.49,328.42,0.00),v40,fine,tPen\WObj:=wPaper;
    MoveL Offs(pOrigin,217.49,328.42,6.00),v60,z5,tPen\WObj:=wPaper;
    MoveL Offs(pOrigin,214.94,332.67,6.00),vTravel,z5,tPen\WObj:=wPaper;
    MoveL Offs(pOrigin,214.94,332.67,0.00),v60,z0,tPen\WObj:=wPaper;
    MoveL Offs(pOrigin,223.01,333.60,0.00),v40,z0,tPen\WObj:=wPaper;
    MoveL Offs(pOrigin,224.50,333.52,0.00),v40,z0,tPen\WObj:=wPaper;
    MoveL Offs(pOrigin,227.26,332.67,0.00),v40,z0,tPen\WObj:=wPaper;
    MoveL Offs(pOrigin,227.26,332.67,0.00),v40,z0,tPen\WObj:=wPaper;
    MoveL Offs(pOrigin,227.48,331.40,0.00),v40,z0,tPen\WObj:=wPaper;
    MoveL Offs(pOrigin,227.05,330.98,0.00),v40,z0,tPen\WObj:=wPaper;
    MoveL Offs(pOrigin,225.35,331.40,0.00),v40,z0,tPen\WObj:=wPaper;
    MoveL Offs(pOrigin,222.59,331.40,0.00),v40,z0,tPen\WObj:=wPaper;
    MoveL Offs(pOrigin,221.74,330.98,0.00),v40,z0,tPen\WObj:=wPaper;
    MoveL Offs(pOrigin,221.74,330.98,0.00),v40,z0,tPen\WObj:=wPaper;
    MoveL Offs(pOrigin,222.02,330.41,0.00),v40,z0,tPen\WObj:=wPaper;
    MoveL Offs(pOrigin,223.86,329.70,0.00),v40,z0,tPen\WObj:=wPaper;
    MoveL Offs(pOrigin,223.44,329.91,0.00),v40,z0,tPen\WObj:=wPaper;
    MoveL Offs(pOrigin,223.86,329.70,0.00),v40,z0,tPen\WObj:=wPaper;
    MoveL Offs(pOrigin,223.44,329.91,0.00),v40,fine,tPen\WObj:=wPaper;
    MoveL Offs(pOrigin,223.44,329.91,6.00),v60,z5,tPen\WObj:=wPaper;
    MoveL Offs(pOrigin,221.74,330.98,6.00),vTravel,z5,tPen\WObj:=wPaper;
    MoveL Offs(pOrigin,221.74,330.98,0.00),v60,z0,tPen\WObj:=wPaper;
    MoveL Offs(pOrigin,216.43,331.19,0.00),v40,z0,tPen\WObj:=wPaper;
    MoveL Offs(pOrigin,214.73,330.98,0.00),v40,z0,tPen\WObj:=wPaper;
    MoveL Offs(pOrigin,210.48,329.49,0.00),v40,z0,tPen\WObj:=wPaper;
    MoveL Offs(pOrigin,209.91,329.70,0.00),v40,z0,tPen\WObj:=wPaper;
    MoveL Offs(pOrigin,210.26,330.34,0.00),v40,z0,tPen\WObj:=wPaper;
    MoveL Offs(pOrigin,211.75,331.33,0.00),v40,z0,tPen\WObj:=wPaper;
    MoveL Offs(pOrigin,214.30,332.11,0.00),v40,z0,tPen\WObj:=wPaper;
    MoveL Offs(pOrigin,214.94,332.67,0.00),v40,fine,tPen\WObj:=wPaper;
    MoveL Offs(pOrigin,214.94,332.67,6.00),v60,z5,tPen\WObj:=wPaper;
    MoveL Offs(pOrigin,211.75,333.52,6.00),vTravel,z5,tPen\WObj:=wPaper;
    MoveL Offs(pOrigin,211.75,333.52,0.00),v60,z0,tPen\WObj:=wPaper;
    MoveL Offs(pOrigin,208.14,331.83,0.00),v40,z0,tPen\WObj:=wPaper;
    MoveL Offs(pOrigin,205.38,329.27,0.00),v40,z0,tPen\WObj:=wPaper;
    MoveL Offs(pOrigin,202.47,325.02,0.00),v40,z0,tPen\WObj:=wPaper;
    MoveL Offs(pOrigin,202.61,323.54,0.00),v40,z0,tPen\WObj:=wPaper;
    MoveL Offs(pOrigin,202.61,323.54,0.00),v40,z0,tPen\WObj:=wPaper;
    MoveL Offs(pOrigin,201.12,321.62,0.00),v40,z0,tPen\WObj:=wPaper;
    MoveL Offs(pOrigin,201.12,321.62,0.00),v40,z0,tPen\WObj:=wPaper;
    MoveL Offs(pOrigin,202.19,321.20,0.00),v40,z0,tPen\WObj:=wPaper;
    MoveL Offs(pOrigin,205.59,322.26,0.00),v40,z0,tPen\WObj:=wPaper;
    MoveL Offs(pOrigin,207.71,322.26,0.00),v40,z0,tPen\WObj:=wPaper;
    MoveL Offs(pOrigin,209.62,321.70,0.00),v40,z0,tPen\WObj:=wPaper;
    MoveL Offs(pOrigin,212.18,319.85,0.00),v40,z0,tPen\WObj:=wPaper;
    MoveL Offs(pOrigin,212.60,320.14,0.00),v40,z0,tPen\WObj:=wPaper;
    MoveL Offs(pOrigin,212.39,321.20,0.00),v40,fine,tPen\WObj:=wPaper;
    MoveL Offs(pOrigin,212.39,321.20,6.00),v60,z5,tPen\WObj:=wPaper;
    MoveL Offs(pOrigin,212.60,323.54,6.00),vTravel,z5,tPen\WObj:=wPaper;
    MoveL Offs(pOrigin,212.60,323.54,0.00),v60,z0,tPen\WObj:=wPaper;
    MoveL Offs(pOrigin,214.09,322.90,0.00),v40,z0,tPen\WObj:=wPaper;
    MoveL Offs(pOrigin,214.58,322.05,0.00),v40,z0,tPen\WObj:=wPaper;
    MoveL Offs(pOrigin,215.36,319.08,0.00),v40,z0,tPen\WObj:=wPaper;
    MoveL Offs(pOrigin,215.36,316.31,0.00),v40,z0,tPen\WObj:=wPaper;
    MoveL Offs(pOrigin,216.57,313.55,0.00),v40,z0,tPen\WObj:=wPaper;
    MoveL Offs(pOrigin,217.06,313.05,0.00),v40,z0,tPen\WObj:=wPaper;
    MoveL Offs(pOrigin,218.34,312.91,0.00),v40,fine,tPen\WObj:=wPaper;
    MoveL Offs(pOrigin,218.34,312.91,6.00),v60,z5,tPen\WObj:=wPaper;
    MoveL Offs(pOrigin,218.76,310.79,6.00),vTravel,z5,tPen\WObj:=wPaper;
    MoveL Offs(pOrigin,218.76,310.79,0.00),v60,z0,tPen\WObj:=wPaper;
    MoveL Offs(pOrigin,218.83,309.51,0.00),v40,z0,tPen\WObj:=wPaper;
    MoveL Offs(pOrigin,219.75,309.02,0.00),v40,z0,tPen\WObj:=wPaper;
    MoveL Offs(pOrigin,219.61,308.73,0.00),v40,z0,tPen\WObj:=wPaper;
    MoveL Offs(pOrigin,218.12,308.66,0.00),v40,z0,tPen\WObj:=wPaper;
    MoveL Offs(pOrigin,216.21,309.51,0.00),v40,fine,tPen\WObj:=wPaper;
    MoveL Offs(pOrigin,216.21,309.51,6.00),v60,z5,tPen\WObj:=wPaper;
    MoveL Offs(pOrigin,216.00,312.06,6.00),vTravel,z5,tPen\WObj:=wPaper;
    MoveL Offs(pOrigin,216.00,312.06,0.00),v60,z0,tPen\WObj:=wPaper;
    MoveL Offs(pOrigin,215.15,312.91,0.00),v40,z0,tPen\WObj:=wPaper;
    MoveL Offs(pOrigin,216.00,312.06,0.00),v40,fine,tPen\WObj:=wPaper;
    MoveL Offs(pOrigin,216.00,312.06,6.00),v60,z5,tPen\WObj:=wPaper;
    MoveL Offs(pOrigin,216.21,313.98,6.00),vTravel,z5,tPen\WObj:=wPaper;
    MoveL Offs(pOrigin,216.21,313.98,0.00),v60,z0,tPen\WObj:=wPaper;
  ENDPROC

  PROC DrawPart41()
    MoveL Offs(pOrigin,216.00,314.40,0.00),v40,z0,tPen\WObj:=wPaper;
    MoveL Offs(pOrigin,216.21,313.98,0.00),v40,fine,tPen\WObj:=wPaper;
    MoveL Offs(pOrigin,216.21,313.98,6.00),v60,z5,tPen\WObj:=wPaper;
    MoveL Offs(pOrigin,218.76,310.79,6.00),vTravel,z5,tPen\WObj:=wPaper;
    MoveL Offs(pOrigin,218.76,310.79,0.00),v60,z0,tPen\WObj:=wPaper;
    MoveL Offs(pOrigin,220.04,310.65,0.00),v40,z0,tPen\WObj:=wPaper;
    MoveL Offs(pOrigin,222.80,309.30,0.00),v40,fine,tPen\WObj:=wPaper;
    MoveL Offs(pOrigin,222.80,309.30,6.00),v60,z5,tPen\WObj:=wPaper;
    MoveL Offs(pOrigin,229.18,319.92,6.00),vTravel,z5,tPen\WObj:=wPaper;
    MoveL Offs(pOrigin,229.18,319.92,0.00),v60,z0,tPen\WObj:=wPaper;
    MoveL Offs(pOrigin,230.24,320.14,0.00),v40,z0,tPen\WObj:=wPaper;
    MoveL Offs(pOrigin,230.24,320.14,0.00),v40,z0,tPen\WObj:=wPaper;
    MoveL Offs(pOrigin,233.28,325.02,0.00),v40,z0,tPen\WObj:=wPaper;
    MoveL Offs(pOrigin,233.64,326.73,0.00),v40,z0,tPen\WObj:=wPaper;
    MoveL Offs(pOrigin,233.07,329.27,0.00),v40,z0,tPen\WObj:=wPaper;
    MoveL Offs(pOrigin,231.73,330.98,0.00),v40,z0,tPen\WObj:=wPaper;
    MoveL Offs(pOrigin,229.81,332.11,0.00),v40,z0,tPen\WObj:=wPaper;
    MoveL Offs(pOrigin,227.26,332.67,0.00),v40,fine,tPen\WObj:=wPaper;
    MoveL Offs(pOrigin,227.26,332.67,6.00),v60,z5,tPen\WObj:=wPaper;
    MoveL Offs(pOrigin,227.48,330.98,6.00),vTravel,z5,tPen\WObj:=wPaper;
    MoveL Offs(pOrigin,227.48,330.98,0.00),v60,z0,tPen\WObj:=wPaper;
    MoveL Offs(pOrigin,228.96,330.20,0.00),v40,z0,tPen\WObj:=wPaper;
    MoveL Offs(pOrigin,229.81,329.27,0.00),v40,z0,tPen\WObj:=wPaper;
    MoveL Offs(pOrigin,230.66,327.15,0.00),v40,z0,tPen\WObj:=wPaper;
    MoveL Offs(pOrigin,230.66,325.02,0.00),v40,z0,tPen\WObj:=wPaper;
    MoveL Offs(pOrigin,228.96,320.77,0.00),v40,z0,tPen\WObj:=wPaper;
    MoveL Offs(pOrigin,229.18,319.92,0.00),v40,z0,tPen\WObj:=wPaper;
    MoveL Offs(pOrigin,230.24,320.14,0.00),v40,z0,tPen\WObj:=wPaper;
    MoveL Offs(pOrigin,231.94,319.92,0.00),v40,z0,tPen\WObj:=wPaper;
    MoveL Offs(pOrigin,231.94,319.92,0.00),v40,z0,tPen\WObj:=wPaper;
    MoveL Offs(pOrigin,234.27,322.05,0.00),v40,fine,tPen\WObj:=wPaper;
    MoveL Offs(pOrigin,234.27,322.05,6.00),v60,z5,tPen\WObj:=wPaper;
    MoveL Offs(pOrigin,233.00,324.17,6.00),vTravel,z5,tPen\WObj:=wPaper;
    MoveL Offs(pOrigin,233.00,324.17,0.00),v60,z0,tPen\WObj:=wPaper;
    MoveL Offs(pOrigin,233.21,324.60,0.00),v40,z0,tPen\WObj:=wPaper;
    MoveL Offs(pOrigin,233.00,324.17,0.00),v40,fine,tPen\WObj:=wPaper;
    MoveL Offs(pOrigin,233.00,324.17,6.00),v60,z5,tPen\WObj:=wPaper;
    MoveL Offs(pOrigin,231.09,321.62,6.00),vTravel,z5,tPen\WObj:=wPaper;
    MoveL Offs(pOrigin,231.09,321.62,0.00),v60,z0,tPen\WObj:=wPaper;
    MoveL Offs(pOrigin,231.73,322.26,0.00),v40,z0,tPen\WObj:=wPaper;
    MoveL Offs(pOrigin,231.09,321.62,0.00),v40,fine,tPen\WObj:=wPaper;
    MoveL Offs(pOrigin,231.09,321.62,6.00),v60,z5,tPen\WObj:=wPaper;
    MoveL Offs(pOrigin,229.60,322.69,6.00),vTravel,z5,tPen\WObj:=wPaper;
    MoveL Offs(pOrigin,229.60,322.69,0.00),v60,z0,tPen\WObj:=wPaper;
    MoveL Offs(pOrigin,229.81,323.11,0.00),v40,z0,tPen\WObj:=wPaper;
    MoveL Offs(pOrigin,229.60,322.69,0.00),v40,fine,tPen\WObj:=wPaper;
    MoveL Offs(pOrigin,229.60,322.69,6.00),v60,z5,tPen\WObj:=wPaper;
    MoveL Offs(pOrigin,229.81,332.25,6.00),vTravel,z5,tPen\WObj:=wPaper;
    MoveL Offs(pOrigin,229.81,332.25,0.00),v60,z0,tPen\WObj:=wPaper;
    MoveL Offs(pOrigin,230.24,332.04,0.00),v40,z0,tPen\WObj:=wPaper;
    MoveL Offs(pOrigin,229.81,332.25,0.00),v40,fine,tPen\WObj:=wPaper;
    MoveL Offs(pOrigin,229.81,332.25,6.00),v60,z5,tPen\WObj:=wPaper;
    MoveL Offs(pOrigin,227.69,337.35,6.00),vTravel,z5,tPen\WObj:=wPaper;
    MoveL Offs(pOrigin,227.69,337.35,0.00),v60,z0,tPen\WObj:=wPaper;
    MoveL Offs(pOrigin,225.56,337.35,0.00),v40,z0,tPen\WObj:=wPaper;
    MoveL Offs(pOrigin,224.93,337.77,0.00),v40,fine,tPen\WObj:=wPaper;
    MoveL Offs(pOrigin,224.93,337.77,6.00),v60,z5,tPen\WObj:=wPaper;
    MoveL Offs(pOrigin,210.69,330.76,6.00),vTravel,z5,tPen\WObj:=wPaper;
    MoveL Offs(pOrigin,210.69,330.76,0.00),v60,z0,tPen\WObj:=wPaper;
    MoveL Offs(pOrigin,211.11,330.98,0.00),v40,z0,tPen\WObj:=wPaper;
    MoveL Offs(pOrigin,210.69,330.76,0.00),v40,fine,tPen\WObj:=wPaper;
    MoveL Offs(pOrigin,210.69,330.76,6.00),v60,z5,tPen\WObj:=wPaper;
    MoveL Offs(pOrigin,209.84,329.49,6.00),vTravel,z5,tPen\WObj:=wPaper;
    MoveL Offs(pOrigin,209.84,329.49,0.00),v60,z0,tPen\WObj:=wPaper;
    MoveL Offs(pOrigin,209.20,329.42,0.00),v40,z0,tPen\WObj:=wPaper;
    MoveL Offs(pOrigin,206.86,327.79,0.00),v40,z0,tPen\WObj:=wPaper;
    MoveL Offs(pOrigin,206.01,325.88,0.00),v40,z0,tPen\WObj:=wPaper;
    MoveL Offs(pOrigin,206.01,325.88,0.00),v40,z0,tPen\WObj:=wPaper;
    MoveL Offs(pOrigin,208.99,326.51,0.00),v40,fine,tPen\WObj:=wPaper;
    MoveL Offs(pOrigin,208.99,326.51,6.00),v60,z5,tPen\WObj:=wPaper;
    MoveL Offs(pOrigin,205.80,325.02,6.00),vTravel,z5,tPen\WObj:=wPaper;
    MoveL Offs(pOrigin,205.80,325.02,0.00),v60,z0,tPen\WObj:=wPaper;
    MoveL Offs(pOrigin,204.52,324.10,0.00),v40,z0,tPen\WObj:=wPaper;
    MoveL Offs(pOrigin,202.61,323.54,0.00),v40,z0,tPen\WObj:=wPaper;
    MoveL Offs(pOrigin,202.61,323.54,0.00),v40,z0,tPen\WObj:=wPaper;
    MoveL Offs(pOrigin,201.76,322.48,0.00),v40,z0,tPen\WObj:=wPaper;
    MoveL Offs(pOrigin,201.12,321.62,0.00),v40,z0,tPen\WObj:=wPaper;
    MoveL Offs(pOrigin,197.51,318.23,0.00),v40,z0,tPen\WObj:=wPaper;
    MoveL Offs(pOrigin,196.80,317.16,0.00),v40,z0,tPen\WObj:=wPaper;
    MoveL Offs(pOrigin,195.46,314.19,0.00),v40,z0,tPen\WObj:=wPaper;
    MoveL Offs(pOrigin,196.02,313.34,0.00),v40,z0,tPen\WObj:=wPaper;
    MoveL Offs(pOrigin,196.02,313.34,0.00),v40,z0,tPen\WObj:=wPaper;
    MoveL Offs(pOrigin,198.79,314.83,0.00),v40,fine,tPen\WObj:=wPaper;
    MoveL Offs(pOrigin,198.79,314.83,6.00),v60,z5,tPen\WObj:=wPaper;
    MoveL Offs(pOrigin,196.02,315.89,6.00),vTravel,z5,tPen\WObj:=wPaper;
    MoveL Offs(pOrigin,196.02,315.89,0.00),v60,z0,tPen\WObj:=wPaper;
    MoveL Offs(pOrigin,196.24,316.31,0.00),v40,z0,tPen\WObj:=wPaper;
    MoveL Offs(pOrigin,196.02,315.89,0.00),v40,z0,tPen\WObj:=wPaper;
    MoveL Offs(pOrigin,196.45,316.74,0.00),v40,z0,tPen\WObj:=wPaper;
    MoveL Offs(pOrigin,196.66,317.16,0.00),v40,z0,tPen\WObj:=wPaper;
    MoveL Offs(pOrigin,196.45,316.74,0.00),v40,fine,tPen\WObj:=wPaper;
    MoveL Offs(pOrigin,196.45,316.74,6.00),v60,z5,tPen\WObj:=wPaper;
    MoveL Offs(pOrigin,195.60,315.04,6.00),vTravel,z5,tPen\WObj:=wPaper;
    MoveL Offs(pOrigin,195.60,315.04,0.00),v60,z0,tPen\WObj:=wPaper;
    MoveL Offs(pOrigin,195.81,315.46,0.00),v40,z0,tPen\WObj:=wPaper;
    MoveL Offs(pOrigin,195.60,315.04,0.00),v40,fine,tPen\WObj:=wPaper;
    MoveL Offs(pOrigin,195.60,315.04,6.00),v60,z5,tPen\WObj:=wPaper;
    MoveL Offs(pOrigin,196.02,313.34,6.00),vTravel,z5,tPen\WObj:=wPaper;
    MoveL Offs(pOrigin,196.02,313.34,0.00),v60,z0,tPen\WObj:=wPaper;
    MoveL Offs(pOrigin,193.83,309.51,0.00),v40,z0,tPen\WObj:=wPaper;
    MoveL Offs(pOrigin,193.48,307.60,0.00),v40,fine,tPen\WObj:=wPaper;
    MoveL Offs(pOrigin,193.48,307.60,6.00),v60,z5,tPen\WObj:=wPaper;
    MoveL Offs(pOrigin,194.11,309.73,6.00),vTravel,z5,tPen\WObj:=wPaper;
    MoveL Offs(pOrigin,194.11,309.73,0.00),v60,z0,tPen\WObj:=wPaper;
    MoveL Offs(pOrigin,194.32,310.15,0.00),v40,z0,tPen\WObj:=wPaper;
    MoveL Offs(pOrigin,194.11,309.73,0.00),v40,fine,tPen\WObj:=wPaper;
    MoveL Offs(pOrigin,194.11,309.73,6.00),v60,z5,tPen\WObj:=wPaper;
    MoveL Offs(pOrigin,198.57,319.50,6.00),vTravel,z5,tPen\WObj:=wPaper;
    MoveL Offs(pOrigin,198.57,319.50,0.00),v60,z0,tPen\WObj:=wPaper;
    MoveL Offs(pOrigin,199.43,320.35,0.00),v40,z0,tPen\WObj:=wPaper;
    MoveL Offs(pOrigin,198.57,319.50,0.00),v40,fine,tPen\WObj:=wPaper;
    MoveL Offs(pOrigin,198.57,319.50,6.00),v60,z5,tPen\WObj:=wPaper;
    MoveL Offs(pOrigin,205.59,324.60,6.00),vTravel,z5,tPen\WObj:=wPaper;
    MoveL Offs(pOrigin,205.59,324.60,0.00),v60,z0,tPen\WObj:=wPaper;
    MoveL Offs(pOrigin,205.80,325.02,0.00),v40,z0,tPen\WObj:=wPaper;
    MoveL Offs(pOrigin,205.59,324.60,0.00),v40,z0,tPen\WObj:=wPaper;
    MoveL Offs(pOrigin,205.80,325.02,0.00),v40,z0,tPen\WObj:=wPaper;
    MoveL Offs(pOrigin,206.65,324.39,0.00),v40,z0,tPen\WObj:=wPaper;
    MoveL Offs(pOrigin,209.62,324.60,0.00),v40,z0,tPen\WObj:=wPaper;
    MoveL Offs(pOrigin,212.18,323.75,0.00),v40,fine,tPen\WObj:=wPaper;
  ENDPROC

  PROC DrawPart42()
    MoveL Offs(pOrigin,212.18,323.75,6.00),v60,z5,tPen\WObj:=wPaper;
    MoveL Offs(pOrigin,241.71,312.91,6.00),vTravel,z5,tPen\WObj:=wPaper;
    MoveL Offs(pOrigin,241.71,312.91,0.00),v60,z0,tPen\WObj:=wPaper;
    MoveL Offs(pOrigin,242.14,312.70,0.00),v40,z0,tPen\WObj:=wPaper;
    MoveL Offs(pOrigin,242.56,311.42,0.00),v40,fine,tPen\WObj:=wPaper;
    MoveL Offs(pOrigin,242.56,311.42,6.00),v60,z5,tPen\WObj:=wPaper;
    MoveL Offs(pOrigin,270.61,315.46,6.00),vTravel,z5,tPen\WObj:=wPaper;
    MoveL Offs(pOrigin,270.61,315.46,0.00),v60,z0,tPen\WObj:=wPaper;
    MoveL Offs(pOrigin,271.04,315.11,0.00),v40,z0,tPen\WObj:=wPaper;
    MoveL Offs(pOrigin,274.01,315.82,0.00),v40,z0,tPen\WObj:=wPaper;
    MoveL Offs(pOrigin,280.60,319.71,0.00),v40,z0,tPen\WObj:=wPaper;
    MoveL Offs(pOrigin,283.58,319.92,0.00),v40,z0,tPen\WObj:=wPaper;
    MoveL Offs(pOrigin,286.12,319.50,0.00),v40,fine,tPen\WObj:=wPaper;
    MoveL Offs(pOrigin,286.12,319.50,6.00),v60,z5,tPen\WObj:=wPaper;
    MoveL Offs(pOrigin,288.89,317.80,6.00),vTravel,z5,tPen\WObj:=wPaper;
    MoveL Offs(pOrigin,288.89,317.80,0.00),v60,z0,tPen\WObj:=wPaper;
    MoveL Offs(pOrigin,287.19,318.65,0.00),v40,z0,tPen\WObj:=wPaper;
    MoveL Offs(pOrigin,285.70,320.77,0.00),v40,z0,tPen\WObj:=wPaper;
    MoveL Offs(pOrigin,283.79,321.84,0.00),v40,fine,tPen\WObj:=wPaper;
    MoveL Offs(pOrigin,283.79,321.84,6.00),v60,z5,tPen\WObj:=wPaper;
    MoveL Offs(pOrigin,288.04,314.83,6.00),vTravel,z5,tPen\WObj:=wPaper;
    MoveL Offs(pOrigin,288.04,314.83,0.00),v60,z0,tPen\WObj:=wPaper;
    MoveL Offs(pOrigin,287.61,315.25,0.00),v40,z0,tPen\WObj:=wPaper;
    MoveL Offs(pOrigin,288.04,314.83,0.00),v40,fine,tPen\WObj:=wPaper;
    MoveL Offs(pOrigin,288.04,314.83,6.00),v60,z5,tPen\WObj:=wPaper;
    MoveL Offs(pOrigin,289.74,315.89,6.00),vTravel,z5,tPen\WObj:=wPaper;
    MoveL Offs(pOrigin,289.74,315.89,0.00),v60,z0,tPen\WObj:=wPaper;
    MoveL Offs(pOrigin,289.52,316.31,0.00),v40,z0,tPen\WObj:=wPaper;
    MoveL Offs(pOrigin,289.74,315.89,0.00),v40,fine,tPen\WObj:=wPaper;
    MoveL Offs(pOrigin,289.74,315.89,6.00),v60,z5,tPen\WObj:=wPaper;
    MoveL Offs(pOrigin,288.25,310.58,6.00),vTravel,z5,tPen\WObj:=wPaper;
    MoveL Offs(pOrigin,288.25,310.58,0.00),v60,z0,tPen\WObj:=wPaper;
    MoveL Offs(pOrigin,287.40,310.58,0.00),v40,z0,tPen\WObj:=wPaper;
    MoveL Offs(pOrigin,286.76,311.21,0.00),v40,z0,tPen\WObj:=wPaper;
    MoveL Offs(pOrigin,286.98,311.00,0.00),v40,fine,tPen\WObj:=wPaper;
    MoveL Offs(pOrigin,286.98,311.00,6.00),v60,z5,tPen\WObj:=wPaper;
    MoveL Offs(pOrigin,288.89,309.51,6.00),vTravel,z5,tPen\WObj:=wPaper;
    MoveL Offs(pOrigin,288.89,309.51,0.00),v60,z0,tPen\WObj:=wPaper;
    MoveL Offs(pOrigin,288.67,309.94,0.00),v40,z0,tPen\WObj:=wPaper;
    MoveL Offs(pOrigin,288.89,309.51,0.00),v40,fine,tPen\WObj:=wPaper;
    MoveL Offs(pOrigin,288.89,309.51,6.00),v60,z5,tPen\WObj:=wPaper;
    MoveL Offs(pOrigin,274.86,327.79,6.00),vTravel,z5,tPen\WObj:=wPaper;
    MoveL Offs(pOrigin,274.86,327.79,0.00),v60,z0,tPen\WObj:=wPaper;
    MoveL Offs(pOrigin,274.01,327.08,0.00),v40,z0,tPen\WObj:=wPaper;
    MoveL Offs(pOrigin,271.89,326.51,0.00),v40,fine,tPen\WObj:=wPaper;
    MoveL Offs(pOrigin,271.89,326.51,6.00),v60,z5,tPen\WObj:=wPaper;
    MoveL Offs(pOrigin,271.89,328.21,6.00),vTravel,z5,tPen\WObj:=wPaper;
    MoveL Offs(pOrigin,271.89,328.21,0.00),v60,z0,tPen\WObj:=wPaper;
    MoveL Offs(pOrigin,273.38,328.21,0.00),v40,z0,tPen\WObj:=wPaper;
    MoveL Offs(pOrigin,274.01,328.64,0.00),v40,fine,tPen\WObj:=wPaper;
    MoveL Offs(pOrigin,274.01,328.64,6.00),v60,z5,tPen\WObj:=wPaper;
    MoveL Offs(pOrigin,271.67,331.61,6.00),vTravel,z5,tPen\WObj:=wPaper;
    MoveL Offs(pOrigin,271.67,331.61,0.00),v60,z0,tPen\WObj:=wPaper;
    MoveL Offs(pOrigin,271.25,332.04,0.00),v40,z0,tPen\WObj:=wPaper;
    MoveL Offs(pOrigin,271.67,331.61,0.00),v40,fine,tPen\WObj:=wPaper;
    MoveL Offs(pOrigin,271.67,331.61,6.00),v60,z5,tPen\WObj:=wPaper;
    MoveL Offs(pOrigin,205.38,276.36,6.00),vTravel,z5,tPen\WObj:=wPaper;
    MoveL Offs(pOrigin,205.38,276.36,0.00),v60,z0,tPen\WObj:=wPaper;
    MoveL Offs(pOrigin,204.88,274.88,0.00),v40,z0,tPen\WObj:=wPaper;
    MoveL Offs(pOrigin,203.89,273.81,0.00),v40,fine,tPen\WObj:=wPaper;
    MoveL Offs(pOrigin,203.89,273.81,6.00),v60,z5,tPen\WObj:=wPaper;
    MoveL Offs(pOrigin,203.68,271.90,6.00),vTravel,z5,tPen\WObj:=wPaper;
    MoveL Offs(pOrigin,203.68,271.90,0.00),v60,z0,tPen\WObj:=wPaper;
    MoveL Offs(pOrigin,204.10,271.48,0.00),v40,z0,tPen\WObj:=wPaper;
    MoveL Offs(pOrigin,204.95,271.48,0.00),v40,fine,tPen\WObj:=wPaper;
    MoveL Offs(pOrigin,204.95,271.48,6.00),v60,z5,tPen\WObj:=wPaper;
    MoveL Offs(pOrigin,200.49,271.26,6.00),vTravel,z5,tPen\WObj:=wPaper;
    MoveL Offs(pOrigin,200.49,271.26,0.00),v60,z0,tPen\WObj:=wPaper;
    MoveL Offs(pOrigin,200.06,271.26,0.00),v40,z0,tPen\WObj:=wPaper;
    MoveL Offs(pOrigin,199.64,269.99,0.00),v40,z0,tPen\WObj:=wPaper;
    MoveL Offs(pOrigin,199.00,269.35,0.00),v40,z0,tPen\WObj:=wPaper;
    MoveL Offs(pOrigin,199.00,269.35,0.00),v40,z0,tPen\WObj:=wPaper;
    MoveL Offs(pOrigin,199.00,268.71,0.00),v40,z0,tPen\WObj:=wPaper;
    MoveL Offs(pOrigin,199.43,268.50,0.00),v40,z0,tPen\WObj:=wPaper;
    MoveL Offs(pOrigin,199.43,268.50,0.00),v40,z0,tPen\WObj:=wPaper;
    MoveL Offs(pOrigin,200.06,269.14,0.00),v40,z0,tPen\WObj:=wPaper;
    MoveL Offs(pOrigin,200.49,269.35,0.00),v40,z0,tPen\WObj:=wPaper;
    MoveL Offs(pOrigin,200.70,269.77,0.00),v40,z0,tPen\WObj:=wPaper;
    MoveL Offs(pOrigin,200.49,269.35,0.00),v40,fine,tPen\WObj:=wPaper;
    MoveL Offs(pOrigin,200.49,269.35,6.00),v60,z5,tPen\WObj:=wPaper;
    MoveL Offs(pOrigin,198.57,273.17,6.00),vTravel,z5,tPen\WObj:=wPaper;
    MoveL Offs(pOrigin,198.57,273.17,0.00),v60,z0,tPen\WObj:=wPaper;
    MoveL Offs(pOrigin,197.94,273.17,0.00),v40,z0,tPen\WObj:=wPaper;
    MoveL Offs(pOrigin,197.51,273.60,0.00),v40,z0,tPen\WObj:=wPaper;
    MoveL Offs(pOrigin,197.51,273.60,0.00),v40,z0,tPen\WObj:=wPaper;
    MoveL Offs(pOrigin,198.15,274.24,0.00),v40,fine,tPen\WObj:=wPaper;
    MoveL Offs(pOrigin,198.15,274.24,6.00),v60,z5,tPen\WObj:=wPaper;
    MoveL Offs(pOrigin,194.32,277.85,6.00),vTravel,z5,tPen\WObj:=wPaper;
    MoveL Offs(pOrigin,194.32,277.85,0.00),v60,z0,tPen\WObj:=wPaper;
    MoveL Offs(pOrigin,193.40,278.49,0.00),v40,z0,tPen\WObj:=wPaper;
    MoveL Offs(pOrigin,193.26,280.19,0.00),v40,z0,tPen\WObj:=wPaper;
    MoveL Offs(pOrigin,193.26,280.19,0.00),v40,z0,tPen\WObj:=wPaper;
    MoveL Offs(pOrigin,193.05,281.25,0.00),v40,z0,tPen\WObj:=wPaper;
    MoveL Offs(pOrigin,193.26,280.19,0.00),v40,z0,tPen\WObj:=wPaper;
    MoveL Offs(pOrigin,195.39,280.19,0.00),v40,fine,tPen\WObj:=wPaper;
    MoveL Offs(pOrigin,195.39,280.19,6.00),v60,z5,tPen\WObj:=wPaper;
    MoveL Offs(pOrigin,197.51,283.38,6.00),vTravel,z5,tPen\WObj:=wPaper;
    MoveL Offs(pOrigin,197.51,283.38,0.00),v60,z0,tPen\WObj:=wPaper;
    MoveL Offs(pOrigin,197.94,283.80,0.00),v40,z0,tPen\WObj:=wPaper;
    MoveL Offs(pOrigin,197.51,283.38,0.00),v40,fine,tPen\WObj:=wPaper;
    MoveL Offs(pOrigin,197.51,283.38,6.00),v60,z5,tPen\WObj:=wPaper;
    MoveL Offs(pOrigin,196.02,285.92,6.00),vTravel,z5,tPen\WObj:=wPaper;
    MoveL Offs(pOrigin,196.02,285.92,0.00),v60,z0,tPen\WObj:=wPaper;
    MoveL Offs(pOrigin,196.24,286.35,0.00),v40,z0,tPen\WObj:=wPaper;
    MoveL Offs(pOrigin,196.02,285.92,0.00),v40,fine,tPen\WObj:=wPaper;
    MoveL Offs(pOrigin,196.02,285.92,6.00),v60,z5,tPen\WObj:=wPaper;
    MoveL Offs(pOrigin,194.32,287.84,6.00),vTravel,z5,tPen\WObj:=wPaper;
    MoveL Offs(pOrigin,194.32,287.84,0.00),v60,z0,tPen\WObj:=wPaper;
    MoveL Offs(pOrigin,191.77,286.35,0.00),v40,fine,tPen\WObj:=wPaper;
    MoveL Offs(pOrigin,191.77,286.35,6.00),v60,z5,tPen\WObj:=wPaper;
    MoveL Offs(pOrigin,196.66,261.70,6.00),vTravel,z5,tPen\WObj:=wPaper;
    MoveL Offs(pOrigin,196.66,261.70,0.00),v60,z0,tPen\WObj:=wPaper;
    MoveL Offs(pOrigin,196.88,262.12,0.00),v40,z0,tPen\WObj:=wPaper;
    MoveL Offs(pOrigin,196.66,261.70,0.00),v40,fine,tPen\WObj:=wPaper;
    MoveL Offs(pOrigin,196.66,261.70,6.00),v60,z5,tPen\WObj:=wPaper;
    MoveL Offs(pOrigin,196.45,251.07,6.00),vTravel,z5,tPen\WObj:=wPaper;
    MoveL Offs(pOrigin,196.45,251.07,0.00),v60,z0,tPen\WObj:=wPaper;
    MoveL Offs(pOrigin,196.24,251.50,0.00),v40,z0,tPen\WObj:=wPaper;
    MoveL Offs(pOrigin,196.45,251.07,0.00),v40,fine,tPen\WObj:=wPaper;
    MoveL Offs(pOrigin,196.45,251.07,6.00),v60,z5,tPen\WObj:=wPaper;
  ENDPROC

  PROC DrawPart43()
    MoveL Offs(pOrigin,227.05,203.69,6.00),vTravel,z5,tPen\WObj:=wPaper;
    MoveL Offs(pOrigin,227.05,203.69,0.00),v60,z0,tPen\WObj:=wPaper;
    MoveL Offs(pOrigin,228.32,203.33,0.00),v40,z0,tPen\WObj:=wPaper;
    MoveL Offs(pOrigin,234.06,199.79,0.00),v40,z0,tPen\WObj:=wPaper;
    MoveL Offs(pOrigin,239.38,197.74,0.00),v40,fine,tPen\WObj:=wPaper;
    MoveL Offs(pOrigin,239.38,197.74,6.00),v60,z5,tPen\WObj:=wPaper;
    MoveL Offs(pOrigin,244.90,198.80,6.00),vTravel,z5,tPen\WObj:=wPaper;
    MoveL Offs(pOrigin,244.90,198.80,0.00),v60,z0,tPen\WObj:=wPaper;
    MoveL Offs(pOrigin,248.09,200.36,0.00),v40,z0,tPen\WObj:=wPaper;
    MoveL Offs(pOrigin,251.06,201.14,0.00),v40,z0,tPen\WObj:=wPaper;
    MoveL Offs(pOrigin,258.29,200.50,0.00),v40,z0,tPen\WObj:=wPaper;
    MoveL Offs(pOrigin,262.11,200.93,0.00),v40,fine,tPen\WObj:=wPaper;
    MoveL Offs(pOrigin,262.11,200.93,6.00),v60,z5,tPen\WObj:=wPaper;
    MoveL Offs(pOrigin,269.76,199.23,6.00),vTravel,z5,tPen\WObj:=wPaper;
    MoveL Offs(pOrigin,269.76,199.23,0.00),v60,z0,tPen\WObj:=wPaper;
    MoveL Offs(pOrigin,273.59,201.56,0.00),v40,z0,tPen\WObj:=wPaper;
    MoveL Offs(pOrigin,278.90,206.02,0.00),v40,z0,tPen\WObj:=wPaper;
    MoveL Offs(pOrigin,280.39,206.66,0.00),v40,fine,tPen\WObj:=wPaper;
    MoveL Offs(pOrigin,280.39,206.66,6.00),v60,z5,tPen\WObj:=wPaper;
    MoveL Offs(pOrigin,282.51,209.85,6.00),vTravel,z5,tPen\WObj:=wPaper;
    MoveL Offs(pOrigin,282.51,209.85,0.00),v60,z0,tPen\WObj:=wPaper;
    MoveL Offs(pOrigin,282.73,210.27,0.00),v40,z0,tPen\WObj:=wPaper;
    MoveL Offs(pOrigin,282.51,209.85,0.00),v40,fine,tPen\WObj:=wPaper;
    MoveL Offs(pOrigin,282.51,209.85,6.00),v60,z5,tPen\WObj:=wPaper;
    MoveL Offs(pOrigin,283.15,211.12,6.00),vTravel,z5,tPen\WObj:=wPaper;
    MoveL Offs(pOrigin,283.15,211.12,0.00),v60,z0,tPen\WObj:=wPaper;
    MoveL Offs(pOrigin,283.36,211.55,0.00),v40,z0,tPen\WObj:=wPaper;
    MoveL Offs(pOrigin,283.15,211.12,0.00),v40,fine,tPen\WObj:=wPaper;
    MoveL Offs(pOrigin,283.15,211.12,6.00),v60,z5,tPen\WObj:=wPaper;
    MoveL Offs(pOrigin,286.76,199.01,6.00),vTravel,z5,tPen\WObj:=wPaper;
    MoveL Offs(pOrigin,286.76,199.01,0.00),v60,z0,tPen\WObj:=wPaper;
    MoveL Offs(pOrigin,287.83,198.73,0.00),v40,z0,tPen\WObj:=wPaper;
    MoveL Offs(pOrigin,289.95,197.31,0.00),v40,z0,tPen\WObj:=wPaper;
    MoveL Offs(pOrigin,294.84,193.06,0.00),v40,z0,tPen\WObj:=wPaper;
    MoveL Offs(pOrigin,300.58,188.95,0.00),v40,z0,tPen\WObj:=wPaper;
    MoveL Offs(pOrigin,302.70,188.46,0.00),v40,z0,tPen\WObj:=wPaper;
    MoveL Offs(pOrigin,303.55,189.31,0.00),v40,z0,tPen\WObj:=wPaper;
    MoveL Offs(pOrigin,312.05,193.20,0.00),v40,z0,tPen\WObj:=wPaper;
    MoveL Offs(pOrigin,314.60,194.76,0.00),v40,z0,tPen\WObj:=wPaper;
    MoveL Offs(pOrigin,314.53,195.61,0.00),v40,z0,tPen\WObj:=wPaper;
    MoveL Offs(pOrigin,308.72,203.05,0.00),v40,z0,tPen\WObj:=wPaper;
    MoveL Offs(pOrigin,308.44,204.32,0.00),v40,fine,tPen\WObj:=wPaper;
    MoveL Offs(pOrigin,308.44,204.32,6.00),v60,z5,tPen\WObj:=wPaper;
    MoveL Offs(pOrigin,309.08,202.62,6.00),vTravel,z5,tPen\WObj:=wPaper;
    MoveL Offs(pOrigin,309.08,202.62,0.00),v60,z0,tPen\WObj:=wPaper;
    MoveL Offs(pOrigin,308.86,203.05,0.00),v40,z0,tPen\WObj:=wPaper;
    MoveL Offs(pOrigin,309.08,202.62,0.00),v40,fine,tPen\WObj:=wPaper;
    MoveL Offs(pOrigin,309.08,202.62,6.00),v60,z5,tPen\WObj:=wPaper;
    MoveL Offs(pOrigin,310.56,200.71,6.00),vTravel,z5,tPen\WObj:=wPaper;
    MoveL Offs(pOrigin,310.56,200.71,0.00),v60,z0,tPen\WObj:=wPaper;
    MoveL Offs(pOrigin,310.35,201.14,0.00),v40,z0,tPen\WObj:=wPaper;
    MoveL Offs(pOrigin,310.56,200.71,0.00),v40,fine,tPen\WObj:=wPaper;
    MoveL Offs(pOrigin,310.56,200.71,6.00),v60,z5,tPen\WObj:=wPaper;
    MoveL Offs(pOrigin,311.41,199.65,6.00),vTravel,z5,tPen\WObj:=wPaper;
    MoveL Offs(pOrigin,311.41,199.65,0.00),v60,z0,tPen\WObj:=wPaper;
    MoveL Offs(pOrigin,311.20,200.07,0.00),v40,z0,tPen\WObj:=wPaper;
    MoveL Offs(pOrigin,311.41,199.65,0.00),v40,z0,tPen\WObj:=wPaper;
    MoveL Offs(pOrigin,311.84,199.23,0.00),v40,z0,tPen\WObj:=wPaper;
    MoveL Offs(pOrigin,312.05,198.80,0.00),v40,z0,tPen\WObj:=wPaper;
    MoveL Offs(pOrigin,311.84,199.23,0.00),v40,fine,tPen\WObj:=wPaper;
    MoveL Offs(pOrigin,311.84,199.23,6.00),v60,z5,tPen\WObj:=wPaper;
    MoveL Offs(pOrigin,315.45,196.68,6.00),vTravel,z5,tPen\WObj:=wPaper;
    MoveL Offs(pOrigin,315.45,196.68,0.00),v60,z0,tPen\WObj:=wPaper;
    MoveL Offs(pOrigin,318.71,191.36,0.00),v40,z0,tPen\WObj:=wPaper;
    MoveL Offs(pOrigin,319.91,188.39,0.00),v40,z0,tPen\WObj:=wPaper;
    MoveL Offs(pOrigin,320.55,185.62,0.00),v40,z0,tPen\WObj:=wPaper;
    MoveL Offs(pOrigin,320.76,183.50,0.00),v40,z0,tPen\WObj:=wPaper;
    MoveL Offs(pOrigin,320.55,179.25,0.00),v40,z0,tPen\WObj:=wPaper;
    MoveL Offs(pOrigin,318.64,172.02,0.00),v40,fine,tPen\WObj:=wPaper;
    MoveL Offs(pOrigin,318.64,172.02,6.00),v60,z5,tPen\WObj:=wPaper;
    MoveL Offs(pOrigin,331.03,172.59,6.00),vTravel,z5,tPen\WObj:=wPaper;
    MoveL Offs(pOrigin,331.03,172.59,0.00),v60,z0,tPen\WObj:=wPaper;
    MoveL Offs(pOrigin,333.73,175.21,0.00),v40,z0,tPen\WObj:=wPaper;
    MoveL Offs(pOrigin,331.03,172.59,0.00),v40,fine,tPen\WObj:=wPaper;
    MoveL Offs(pOrigin,331.03,172.59,6.00),v60,z5,tPen\WObj:=wPaper;
    MoveL Offs(pOrigin,334.15,175.64,6.00),vTravel,z5,tPen\WObj:=wPaper;
    MoveL Offs(pOrigin,334.15,175.64,0.00),v60,z0,tPen\WObj:=wPaper;
    MoveL Offs(pOrigin,334.58,176.06,0.00),v40,z0,tPen\WObj:=wPaper;
    MoveL Offs(pOrigin,334.15,175.64,0.00),v40,fine,tPen\WObj:=wPaper;
    MoveL Offs(pOrigin,334.15,175.64,6.00),v60,z5,tPen\WObj:=wPaper;
    MoveL Offs(pOrigin,340.31,180.95,6.00),vTravel,z5,tPen\WObj:=wPaper;
    MoveL Offs(pOrigin,340.31,180.95,0.00),v60,z0,tPen\WObj:=wPaper;
    MoveL Offs(pOrigin,334.36,176.06,0.00),v40,z0,tPen\WObj:=wPaper;
    MoveL Offs(pOrigin,330.75,172.45,0.00),v40,z0,tPen\WObj:=wPaper;
    MoveL Offs(pOrigin,323.74,164.16,0.00),v40,z0,tPen\WObj:=wPaper;
    MoveL Offs(pOrigin,314.95,151.20,0.00),v40,z0,tPen\WObj:=wPaper;
    MoveL Offs(pOrigin,310.14,141.85,0.00),v40,fine,tPen\WObj:=wPaper;
    MoveL Offs(pOrigin,310.14,141.85,6.00),v60,z5,tPen\WObj:=wPaper;
    MoveL Offs(pOrigin,310.77,143.12,6.00),vTravel,z5,tPen\WObj:=wPaper;
    MoveL Offs(pOrigin,310.77,143.12,0.00),v60,z0,tPen\WObj:=wPaper;
    MoveL Offs(pOrigin,310.99,143.55,0.00),v40,z0,tPen\WObj:=wPaper;
    MoveL Offs(pOrigin,310.77,143.12,0.00),v40,fine,tPen\WObj:=wPaper;
    MoveL Offs(pOrigin,310.77,143.12,6.00),v60,z5,tPen\WObj:=wPaper;
    MoveL Offs(pOrigin,313.33,148.01,6.00),vTravel,z5,tPen\WObj:=wPaper;
    MoveL Offs(pOrigin,313.33,148.01,0.00),v60,z0,tPen\WObj:=wPaper;
    MoveL Offs(pOrigin,313.54,148.44,0.00),v40,z0,tPen\WObj:=wPaper;
    MoveL Offs(pOrigin,313.33,148.01,0.00),v40,fine,tPen\WObj:=wPaper;
    MoveL Offs(pOrigin,313.33,148.01,6.00),v60,z5,tPen\WObj:=wPaper;
    MoveL Offs(pOrigin,314.17,149.50,6.00),vTravel,z5,tPen\WObj:=wPaper;
    MoveL Offs(pOrigin,314.17,149.50,0.00),v60,z0,tPen\WObj:=wPaper;
    MoveL Offs(pOrigin,314.39,149.93,0.00),v40,z0,tPen\WObj:=wPaper;
    MoveL Offs(pOrigin,314.17,149.50,0.00),v40,fine,tPen\WObj:=wPaper;
    MoveL Offs(pOrigin,314.17,149.50,6.00),v60,z5,tPen\WObj:=wPaper;
    MoveL Offs(pOrigin,314.81,150.56,6.00),vTravel,z5,tPen\WObj:=wPaper;
    MoveL Offs(pOrigin,314.81,150.56,0.00),v60,z0,tPen\WObj:=wPaper;
    MoveL Offs(pOrigin,315.02,150.99,0.00),v40,z0,tPen\WObj:=wPaper;
    MoveL Offs(pOrigin,314.81,150.56,0.00),v40,fine,tPen\WObj:=wPaper;
    MoveL Offs(pOrigin,314.81,150.56,6.00),v60,z5,tPen\WObj:=wPaper;
    MoveL Offs(pOrigin,305.46,169.05,6.00),vTravel,z5,tPen\WObj:=wPaper;
    MoveL Offs(pOrigin,305.46,169.05,0.00),v60,z0,tPen\WObj:=wPaper;
    MoveL Offs(pOrigin,302.91,169.83,0.00),v40,z0,tPen\WObj:=wPaper;
    MoveL Offs(pOrigin,297.39,172.17,0.00),v40,z0,tPen\WObj:=wPaper;
    MoveL Offs(pOrigin,296.82,173.02,0.00),v40,z0,tPen\WObj:=wPaper;
    MoveL Offs(pOrigin,297.60,173.09,0.00),v40,z0,tPen\WObj:=wPaper;
    MoveL Offs(pOrigin,305.67,170.18,0.00),v40,z0,tPen\WObj:=wPaper;
    MoveL Offs(pOrigin,306.03,169.48,0.00),v40,z0,tPen\WObj:=wPaper;
    MoveL Offs(pOrigin,305.46,169.05,0.00),v40,fine,tPen\WObj:=wPaper;
    MoveL Offs(pOrigin,305.46,169.05,6.00),v60,z5,tPen\WObj:=wPaper;
    MoveL Offs(pOrigin,297.17,172.45,6.00),vTravel,z5,tPen\WObj:=wPaper;
    MoveL Offs(pOrigin,297.17,172.45,0.00),v60,z0,tPen\WObj:=wPaper;
  ENDPROC

  PROC DrawPart44()
    MoveL Offs(pOrigin,297.60,172.24,0.00),v40,z0,tPen\WObj:=wPaper;
    MoveL Offs(pOrigin,297.17,172.45,0.00),v40,z0,tPen\WObj:=wPaper;
    MoveL Offs(pOrigin,296.75,173.09,0.00),v40,z0,tPen\WObj:=wPaper;
    MoveL Offs(pOrigin,295.69,173.30,0.00),v40,fine,tPen\WObj:=wPaper;
    MoveL Offs(pOrigin,295.69,173.30,6.00),v60,z5,tPen\WObj:=wPaper;
    MoveL Offs(pOrigin,280.39,175.85,6.00),vTravel,z5,tPen\WObj:=wPaper;
    MoveL Offs(pOrigin,280.39,175.85,0.00),v60,z0,tPen\WObj:=wPaper;
    MoveL Offs(pOrigin,279.47,176.49,0.00),v40,z0,tPen\WObj:=wPaper;
    MoveL Offs(pOrigin,278.26,181.38,0.00),v40,z0,tPen\WObj:=wPaper;
    MoveL Offs(pOrigin,277.84,181.59,0.00),v40,z0,tPen\WObj:=wPaper;
    MoveL Offs(pOrigin,277.84,181.59,0.00),v40,z0,tPen\WObj:=wPaper;
    MoveL Offs(pOrigin,277.84,183.29,0.00),v40,z0,tPen\WObj:=wPaper;
    MoveL Offs(pOrigin,277.41,184.99,0.00),v40,z0,tPen\WObj:=wPaper;
    MoveL Offs(pOrigin,275.92,187.96,0.00),v40,z0,tPen\WObj:=wPaper;
    MoveL Offs(pOrigin,275.50,188.18,0.00),v40,z0,tPen\WObj:=wPaper;
    MoveL Offs(pOrigin,274.01,188.60,0.00),v40,z0,tPen\WObj:=wPaper;
    MoveL Offs(pOrigin,272.31,187.54,0.00),v40,z0,tPen\WObj:=wPaper;
    MoveL Offs(pOrigin,267.00,178.82,0.00),v40,fine,tPen\WObj:=wPaper;
    MoveL Offs(pOrigin,267.00,178.82,6.00),v60,z5,tPen\WObj:=wPaper;
    MoveL Offs(pOrigin,268.06,176.06,6.00),vTravel,z5,tPen\WObj:=wPaper;
    MoveL Offs(pOrigin,268.06,176.06,0.00),v60,z0,tPen\WObj:=wPaper;
    MoveL Offs(pOrigin,271.89,177.90,0.00),v40,z0,tPen\WObj:=wPaper;
    MoveL Offs(pOrigin,277.20,181.45,0.00),v40,z0,tPen\WObj:=wPaper;
    MoveL Offs(pOrigin,277.84,181.59,0.00),v40,fine,tPen\WObj:=wPaper;
    MoveL Offs(pOrigin,277.84,181.59,6.00),v60,z5,tPen\WObj:=wPaper;
    MoveL Offs(pOrigin,277.62,178.19,6.00),vTravel,z5,tPen\WObj:=wPaper;
    MoveL Offs(pOrigin,277.62,178.19,0.00),v60,z0,tPen\WObj:=wPaper;
    MoveL Offs(pOrigin,271.82,165.44,0.00),v40,z0,tPen\WObj:=wPaper;
    MoveL Offs(pOrigin,269.98,160.55,0.00),v40,fine,tPen\WObj:=wPaper;
    MoveL Offs(pOrigin,269.98,160.55,6.00),v60,z5,tPen\WObj:=wPaper;
    MoveL Offs(pOrigin,272.10,166.29,6.00),vTravel,z5,tPen\WObj:=wPaper;
    MoveL Offs(pOrigin,272.10,166.29,0.00),v60,z0,tPen\WObj:=wPaper;
    MoveL Offs(pOrigin,272.31,166.71,0.00),v40,z0,tPen\WObj:=wPaper;
    MoveL Offs(pOrigin,272.10,166.29,0.00),v40,fine,tPen\WObj:=wPaper;
    MoveL Offs(pOrigin,272.10,166.29,6.00),v60,z5,tPen\WObj:=wPaper;
    MoveL Offs(pOrigin,272.74,167.77,6.00),vTravel,z5,tPen\WObj:=wPaper;
    MoveL Offs(pOrigin,272.74,167.77,0.00),v60,z0,tPen\WObj:=wPaper;
    MoveL Offs(pOrigin,272.95,168.20,0.00),v40,z0,tPen\WObj:=wPaper;
    MoveL Offs(pOrigin,272.74,167.77,0.00),v40,fine,tPen\WObj:=wPaper;
    MoveL Offs(pOrigin,272.74,167.77,6.00),v60,z5,tPen\WObj:=wPaper;
    MoveL Offs(pOrigin,274.86,172.45,6.00),vTravel,z5,tPen\WObj:=wPaper;
    MoveL Offs(pOrigin,274.86,172.45,0.00),v60,z0,tPen\WObj:=wPaper;
    MoveL Offs(pOrigin,275.08,172.88,0.00),v40,z0,tPen\WObj:=wPaper;
    MoveL Offs(pOrigin,274.86,172.45,0.00),v40,fine,tPen\WObj:=wPaper;
    MoveL Offs(pOrigin,274.86,172.45,6.00),v60,z5,tPen\WObj:=wPaper;
    MoveL Offs(pOrigin,274.23,174.79,6.00),vTravel,z5,tPen\WObj:=wPaper;
    MoveL Offs(pOrigin,274.23,174.79,0.00),v60,z0,tPen\WObj:=wPaper;
    MoveL Offs(pOrigin,275.50,176.49,0.00),v40,fine,tPen\WObj:=wPaper;
    MoveL Offs(pOrigin,275.50,176.49,6.00),v60,z5,tPen\WObj:=wPaper;
    MoveL Offs(pOrigin,268.06,173.73,6.00),vTravel,z5,tPen\WObj:=wPaper;
    MoveL Offs(pOrigin,268.06,173.73,0.00),v60,z0,tPen\WObj:=wPaper;
    MoveL Offs(pOrigin,266.36,171.18,0.00),v40,z0,tPen\WObj:=wPaper;
    MoveL Offs(pOrigin,263.60,167.99,0.00),v40,z0,tPen\WObj:=wPaper;
    MoveL Offs(pOrigin,257.01,162.46,0.00),v40,fine,tPen\WObj:=wPaper;
    MoveL Offs(pOrigin,257.01,162.46,6.00),v60,z5,tPen\WObj:=wPaper;
    MoveL Offs(pOrigin,254.89,155.31,6.00),vTravel,z5,tPen\WObj:=wPaper;
    MoveL Offs(pOrigin,254.89,155.31,0.00),v60,z0,tPen\WObj:=wPaper;
    MoveL Offs(pOrigin,255.60,154.60,0.00),v40,z0,tPen\WObj:=wPaper;
    MoveL Offs(pOrigin,256.16,153.11,0.00),v40,z0,tPen\WObj:=wPaper;
    MoveL Offs(pOrigin,255.81,151.41,0.00),v40,z0,tPen\WObj:=wPaper;
    MoveL Offs(pOrigin,255.10,150.56,0.00),v40,z0,tPen\WObj:=wPaper;
    MoveL Offs(pOrigin,253.61,149.93,0.00),v40,z0,tPen\WObj:=wPaper;
    MoveL Offs(pOrigin,252.12,150.28,0.00),v40,z0,tPen\WObj:=wPaper;
    MoveL Offs(pOrigin,250.78,151.62,0.00),v40,z0,tPen\WObj:=wPaper;
    MoveL Offs(pOrigin,250.43,152.69,0.00),v40,z0,tPen\WObj:=wPaper;
    MoveL Offs(pOrigin,250.78,154.18,0.00),v40,z0,tPen\WObj:=wPaper;
    MoveL Offs(pOrigin,251.70,155.24,0.00),v40,z0,tPen\WObj:=wPaper;
    MoveL Offs(pOrigin,253.19,155.88,0.00),v40,z0,tPen\WObj:=wPaper;
    MoveL Offs(pOrigin,254.89,155.31,0.00),v40,fine,tPen\WObj:=wPaper;
    MoveL Offs(pOrigin,254.89,155.31,6.00),v60,z5,tPen\WObj:=wPaper;
    MoveL Offs(pOrigin,250.85,153.96,6.00),vTravel,z5,tPen\WObj:=wPaper;
    MoveL Offs(pOrigin,250.85,153.96,0.00),v60,z0,tPen\WObj:=wPaper;
    MoveL Offs(pOrigin,251.91,155.24,0.00),v40,z0,tPen\WObj:=wPaper;
    MoveL Offs(pOrigin,250.85,153.96,0.00),v40,fine,tPen\WObj:=wPaper;
    MoveL Offs(pOrigin,250.85,153.96,6.00),v60,z5,tPen\WObj:=wPaper;
    MoveL Offs(pOrigin,251.91,150.56,6.00),vTravel,z5,tPen\WObj:=wPaper;
    MoveL Offs(pOrigin,251.91,150.56,0.00),v60,z0,tPen\WObj:=wPaper;
    MoveL Offs(pOrigin,252.34,150.35,0.00),v40,z0,tPen\WObj:=wPaper;
    MoveL Offs(pOrigin,251.91,150.56,0.00),v40,fine,tPen\WObj:=wPaper;
    MoveL Offs(pOrigin,251.91,150.56,6.00),v60,z5,tPen\WObj:=wPaper;
    MoveL Offs(pOrigin,238.74,143.55,6.00),vTravel,z5,tPen\WObj:=wPaper;
    MoveL Offs(pOrigin,238.74,143.55,0.00),v60,z0,tPen\WObj:=wPaper;
    MoveL Offs(pOrigin,229.32,166.71,0.00),v40,z0,tPen\WObj:=wPaper;
    MoveL Offs(pOrigin,228.11,167.56,0.00),v40,fine,tPen\WObj:=wPaper;
    MoveL Offs(pOrigin,228.11,167.56,6.00),v60,z5,tPen\WObj:=wPaper;
    MoveL Offs(pOrigin,231.30,161.61,6.00),vTravel,z5,tPen\WObj:=wPaper;
    MoveL Offs(pOrigin,231.30,161.61,0.00),v60,z0,tPen\WObj:=wPaper;
    MoveL Offs(pOrigin,231.09,162.04,0.00),v40,z0,tPen\WObj:=wPaper;
    MoveL Offs(pOrigin,231.30,161.61,0.00),v40,z0,tPen\WObj:=wPaper;
    MoveL Offs(pOrigin,231.73,160.55,0.00),v40,z0,tPen\WObj:=wPaper;
    MoveL Offs(pOrigin,231.51,160.98,0.00),v40,z0,tPen\WObj:=wPaper;
    MoveL Offs(pOrigin,231.73,160.55,0.00),v40,fine,tPen\WObj:=wPaper;
    MoveL Offs(pOrigin,231.73,160.55,6.00),v60,z5,tPen\WObj:=wPaper;
    MoveL Offs(pOrigin,234.27,154.39,6.00),vTravel,z5,tPen\WObj:=wPaper;
    MoveL Offs(pOrigin,234.27,154.39,0.00),v60,z0,tPen\WObj:=wPaper;
    MoveL Offs(pOrigin,234.06,154.81,0.00),v40,z0,tPen\WObj:=wPaper;
    MoveL Offs(pOrigin,234.27,154.39,0.00),v40,fine,tPen\WObj:=wPaper;
    MoveL Offs(pOrigin,234.27,154.39,6.00),v60,z5,tPen\WObj:=wPaper;
    MoveL Offs(pOrigin,234.91,152.90,6.00),vTravel,z5,tPen\WObj:=wPaper;
    MoveL Offs(pOrigin,234.91,152.90,0.00),v60,z0,tPen\WObj:=wPaper;
    MoveL Offs(pOrigin,234.70,153.32,0.00),v40,z0,tPen\WObj:=wPaper;
    MoveL Offs(pOrigin,234.91,152.90,0.00),v40,z0,tPen\WObj:=wPaper;
    MoveL Offs(pOrigin,235.34,151.84,0.00),v40,z0,tPen\WObj:=wPaper;
    MoveL Offs(pOrigin,235.12,152.26,0.00),v40,z0,tPen\WObj:=wPaper;
    MoveL Offs(pOrigin,235.34,151.84,0.00),v40,z0,tPen\WObj:=wPaper;
    MoveL Offs(pOrigin,235.76,150.77,0.00),v40,z0,tPen\WObj:=wPaper;
    MoveL Offs(pOrigin,235.55,151.20,0.00),v40,z0,tPen\WObj:=wPaper;
    MoveL Offs(pOrigin,235.76,150.77,0.00),v40,fine,tPen\WObj:=wPaper;
    MoveL Offs(pOrigin,235.76,150.77,6.00),v60,z5,tPen\WObj:=wPaper;
    MoveL Offs(pOrigin,242.56,163.95,6.00),vTravel,z5,tPen\WObj:=wPaper;
    MoveL Offs(pOrigin,242.56,163.95,0.00),v60,z0,tPen\WObj:=wPaper;
    MoveL Offs(pOrigin,241.50,165.44,0.00),v40,z0,tPen\WObj:=wPaper;
    MoveL Offs(pOrigin,241.71,165.01,0.00),v40,z0,tPen\WObj:=wPaper;
    MoveL Offs(pOrigin,241.50,165.44,0.00),v40,z0,tPen\WObj:=wPaper;
    MoveL Offs(pOrigin,241.71,165.01,0.00),v40,fine,tPen\WObj:=wPaper;
    MoveL Offs(pOrigin,241.71,165.01,6.00),v60,z5,tPen\WObj:=wPaper;
    MoveL Offs(pOrigin,238.10,186.90,6.00),vTravel,z5,tPen\WObj:=wPaper;
    MoveL Offs(pOrigin,238.10,186.90,0.00),v60,z0,tPen\WObj:=wPaper;
    MoveL Offs(pOrigin,236.40,188.39,0.00),v40,z0,tPen\WObj:=wPaper;
    MoveL Offs(pOrigin,232.01,194.55,0.00),v40,z0,tPen\WObj:=wPaper;
  ENDPROC

  PROC DrawPart45()
    MoveL Offs(pOrigin,231.73,195.61,0.00),v40,fine,tPen\WObj:=wPaper;
    MoveL Offs(pOrigin,231.73,195.61,6.00),v60,z5,tPen\WObj:=wPaper;
    MoveL Offs(pOrigin,230.66,196.89,6.00),vTravel,z5,tPen\WObj:=wPaper;
    MoveL Offs(pOrigin,230.66,196.89,0.00),v60,z0,tPen\WObj:=wPaper;
    MoveL Offs(pOrigin,230.45,197.31,0.00),v40,z0,tPen\WObj:=wPaper;
    MoveL Offs(pOrigin,230.66,196.89,0.00),v40,fine,tPen\WObj:=wPaper;
    MoveL Offs(pOrigin,230.66,196.89,6.00),v60,z5,tPen\WObj:=wPaper;
    MoveL Offs(pOrigin,227.05,203.69,6.00),vTravel,z5,tPen\WObj:=wPaper;
    MoveL Offs(pOrigin,227.05,203.69,0.00),v60,z0,tPen\WObj:=wPaper;
    MoveL Offs(pOrigin,227.33,202.20,0.00),v40,z0,tPen\WObj:=wPaper;
    MoveL Offs(pOrigin,228.47,200.29,0.00),v40,z0,tPen\WObj:=wPaper;
    MoveL Offs(pOrigin,231.73,195.82,0.00),v40,z0,tPen\WObj:=wPaper;
    MoveL Offs(pOrigin,233.00,195.47,0.00),v40,z0,tPen\WObj:=wPaper;
    MoveL Offs(pOrigin,235.34,193.84,0.00),v40,z0,tPen\WObj:=wPaper;
    MoveL Offs(pOrigin,238.52,192.35,0.00),v40,z0,tPen\WObj:=wPaper;
    MoveL Offs(pOrigin,241.71,191.36,0.00),v40,z0,tPen\WObj:=wPaper;
    MoveL Offs(pOrigin,244.69,190.94,0.00),v40,fine,tPen\WObj:=wPaper;
    MoveL Offs(pOrigin,244.69,190.94,6.00),v60,z5,tPen\WObj:=wPaper;
    MoveL Offs(pOrigin,253.19,191.79,6.00),vTravel,z5,tPen\WObj:=wPaper;
    MoveL Offs(pOrigin,253.19,191.79,0.00),v60,z0,tPen\WObj:=wPaper;
    MoveL Offs(pOrigin,258.08,190.94,0.00),v40,z0,tPen\WObj:=wPaper;
    MoveL Offs(pOrigin,262.54,191.57,0.00),v40,z0,tPen\WObj:=wPaper;
    MoveL Offs(pOrigin,266.58,192.99,0.00),v40,z0,tPen\WObj:=wPaper;
    MoveL Offs(pOrigin,269.98,194.69,0.00),v40,z0,tPen\WObj:=wPaper;
    MoveL Offs(pOrigin,274.01,197.38,0.00),v40,z0,tPen\WObj:=wPaper;
    MoveL Offs(pOrigin,275.29,197.74,0.00),v40,fine,tPen\WObj:=wPaper;
    MoveL Offs(pOrigin,275.29,197.74,6.00),v60,z5,tPen\WObj:=wPaper;
    MoveL Offs(pOrigin,276.35,199.01,6.00),vTravel,z5,tPen\WObj:=wPaper;
    MoveL Offs(pOrigin,276.35,199.01,0.00),v60,z0,tPen\WObj:=wPaper;
    MoveL Offs(pOrigin,276.56,199.44,0.00),v40,z0,tPen\WObj:=wPaper;
    MoveL Offs(pOrigin,276.35,199.01,0.00),v40,fine,tPen\WObj:=wPaper;
    MoveL Offs(pOrigin,276.35,199.01,6.00),v60,z5,tPen\WObj:=wPaper;
    MoveL Offs(pOrigin,269.55,188.81,6.00),vTravel,z5,tPen\WObj:=wPaper;
    MoveL Offs(pOrigin,269.55,188.81,0.00),v60,z0,tPen\WObj:=wPaper;
    MoveL Offs(pOrigin,268.49,188.67,0.00),v40,z0,tPen\WObj:=wPaper;
    MoveL Offs(pOrigin,265.09,186.76,0.00),v40,z0,tPen\WObj:=wPaper;
    MoveL Offs(pOrigin,261.48,185.41,0.00),v40,fine,tPen\WObj:=wPaper;
    MoveL Offs(pOrigin,261.48,185.41,6.00),v60,z5,tPen\WObj:=wPaper;
    MoveL Offs(pOrigin,267.42,188.18,6.00),vTravel,z5,tPen\WObj:=wPaper;
    MoveL Offs(pOrigin,267.42,188.18,0.00),v60,z0,tPen\WObj:=wPaper;
    MoveL Offs(pOrigin,267.85,188.39,0.00),v40,z0,tPen\WObj:=wPaper;
    MoveL Offs(pOrigin,267.42,188.18,0.00),v40,fine,tPen\WObj:=wPaper;
    MoveL Offs(pOrigin,267.42,188.18,6.00),v60,z5,tPen\WObj:=wPaper;
    MoveL Offs(pOrigin,270.61,184.77,6.00),vTravel,z5,tPen\WObj:=wPaper;
    MoveL Offs(pOrigin,270.61,184.77,0.00),v60,z0,tPen\WObj:=wPaper;
    MoveL Offs(pOrigin,270.83,185.20,0.00),v40,z0,tPen\WObj:=wPaper;
    MoveL Offs(pOrigin,270.61,184.77,0.00),v40,fine,tPen\WObj:=wPaper;
    MoveL Offs(pOrigin,270.61,184.77,6.00),v60,z5,tPen\WObj:=wPaper;
    MoveL Offs(pOrigin,264.45,168.84,6.00),vTravel,z5,tPen\WObj:=wPaper;
    MoveL Offs(pOrigin,264.45,168.84,0.00),v60,z0,tPen\WObj:=wPaper;
    MoveL Offs(pOrigin,265.09,169.48,0.00),v40,z0,tPen\WObj:=wPaper;
    MoveL Offs(pOrigin,264.45,168.84,0.00),v40,fine,tPen\WObj:=wPaper;
    MoveL Offs(pOrigin,264.45,168.84,6.00),v60,z5,tPen\WObj:=wPaper;
    MoveL Offs(pOrigin,275.71,152.69,6.00),vTravel,z5,tPen\WObj:=wPaper;
    MoveL Offs(pOrigin,275.71,152.69,0.00),v60,z0,tPen\WObj:=wPaper;
    MoveL Offs(pOrigin,274.51,151.84,0.00),v40,z0,tPen\WObj:=wPaper;
    MoveL Offs(pOrigin,268.70,137.18,0.00),v40,fine,tPen\WObj:=wPaper;
    MoveL Offs(pOrigin,268.70,137.18,6.00),v60,z5,tPen\WObj:=wPaper;
    MoveL Offs(pOrigin,271.67,145.25,6.00),vTravel,z5,tPen\WObj:=wPaper;
    MoveL Offs(pOrigin,271.67,145.25,0.00),v60,z0,tPen\WObj:=wPaper;
    MoveL Offs(pOrigin,271.89,145.68,0.00),v40,z0,tPen\WObj:=wPaper;
    MoveL Offs(pOrigin,271.67,145.25,0.00),v40,fine,tPen\WObj:=wPaper;
    MoveL Offs(pOrigin,271.67,145.25,6.00),v60,z5,tPen\WObj:=wPaper;
    MoveL Offs(pOrigin,268.70,115.07,6.00),vTravel,z5,tPen\WObj:=wPaper;
    MoveL Offs(pOrigin,268.70,115.07,0.00),v60,z0,tPen\WObj:=wPaper;
    MoveL Offs(pOrigin,265.58,107.00,0.00),v40,z0,tPen\WObj:=wPaper;
    MoveL Offs(pOrigin,262.18,99.35,0.00),v40,z0,tPen\WObj:=wPaper;
    MoveL Offs(pOrigin,255.10,85.96,0.00),v40,fine,tPen\WObj:=wPaper;
    MoveL Offs(pOrigin,255.10,85.96,6.00),v60,z5,tPen\WObj:=wPaper;
    MoveL Offs(pOrigin,258.29,92.12,6.00),vTravel,z5,tPen\WObj:=wPaper;
    MoveL Offs(pOrigin,258.29,92.12,0.00),v60,z0,tPen\WObj:=wPaper;
    MoveL Offs(pOrigin,258.50,92.55,0.00),v40,z0,tPen\WObj:=wPaper;
    MoveL Offs(pOrigin,258.29,92.12,0.00),v40,z0,tPen\WObj:=wPaper;
    MoveL Offs(pOrigin,258.71,92.76,0.00),v40,z0,tPen\WObj:=wPaper;
    MoveL Offs(pOrigin,258.92,93.19,0.00),v40,z0,tPen\WObj:=wPaper;
    MoveL Offs(pOrigin,258.71,92.76,0.00),v40,z0,tPen\WObj:=wPaper;
    MoveL Offs(pOrigin,259.14,93.61,0.00),v40,z0,tPen\WObj:=wPaper;
    MoveL Offs(pOrigin,259.35,94.04,0.00),v40,z0,tPen\WObj:=wPaper;
    MoveL Offs(pOrigin,259.14,93.61,0.00),v40,z0,tPen\WObj:=wPaper;
    MoveL Offs(pOrigin,259.56,94.46,0.00),v40,z0,tPen\WObj:=wPaper;
    MoveL Offs(pOrigin,259.77,94.89,0.00),v40,z0,tPen\WObj:=wPaper;
    MoveL Offs(pOrigin,259.56,94.46,0.00),v40,z0,tPen\WObj:=wPaper;
    MoveL Offs(pOrigin,259.99,95.31,0.00),v40,z0,tPen\WObj:=wPaper;
    MoveL Offs(pOrigin,260.20,95.74,0.00),v40,z0,tPen\WObj:=wPaper;
    MoveL Offs(pOrigin,259.99,95.31,0.00),v40,fine,tPen\WObj:=wPaper;
    MoveL Offs(pOrigin,259.99,95.31,6.00),v60,z5,tPen\WObj:=wPaper;
    MoveL Offs(pOrigin,261.90,99.14,6.00),vTravel,z5,tPen\WObj:=wPaper;
    MoveL Offs(pOrigin,261.90,99.14,0.00),v60,z0,tPen\WObj:=wPaper;
    MoveL Offs(pOrigin,262.11,99.56,0.00),v40,z0,tPen\WObj:=wPaper;
    MoveL Offs(pOrigin,261.90,99.14,0.00),v40,fine,tPen\WObj:=wPaper;
    MoveL Offs(pOrigin,261.90,99.14,6.00),v60,z5,tPen\WObj:=wPaper;
    MoveL Offs(pOrigin,262.96,101.47,6.00),vTravel,z5,tPen\WObj:=wPaper;
    MoveL Offs(pOrigin,262.96,101.47,0.00),v60,z0,tPen\WObj:=wPaper;
    MoveL Offs(pOrigin,263.17,101.90,0.00),v40,z0,tPen\WObj:=wPaper;
    MoveL Offs(pOrigin,262.96,101.47,0.00),v40,fine,tPen\WObj:=wPaper;
    MoveL Offs(pOrigin,262.96,101.47,6.00),v60,z5,tPen\WObj:=wPaper;
    MoveL Offs(pOrigin,264.02,103.81,6.00),vTravel,z5,tPen\WObj:=wPaper;
    MoveL Offs(pOrigin,264.02,103.81,0.00),v60,z0,tPen\WObj:=wPaper;
    MoveL Offs(pOrigin,264.24,104.24,0.00),v40,z0,tPen\WObj:=wPaper;
    MoveL Offs(pOrigin,264.02,103.81,0.00),v40,z0,tPen\WObj:=wPaper;
    MoveL Offs(pOrigin,264.45,104.88,0.00),v40,z0,tPen\WObj:=wPaper;
    MoveL Offs(pOrigin,264.66,105.30,0.00),v40,z0,tPen\WObj:=wPaper;
    MoveL Offs(pOrigin,264.45,104.88,0.00),v40,fine,tPen\WObj:=wPaper;
    MoveL Offs(pOrigin,264.45,104.88,6.00),v60,z5,tPen\WObj:=wPaper;
    MoveL Offs(pOrigin,253.19,111.04,6.00),vTravel,z5,tPen\WObj:=wPaper;
    MoveL Offs(pOrigin,253.19,111.04,0.00),v60,z0,tPen\WObj:=wPaper;
    MoveL Offs(pOrigin,251.70,110.40,0.00),v40,z0,tPen\WObj:=wPaper;
    MoveL Offs(pOrigin,250.43,110.40,0.00),v40,z0,tPen\WObj:=wPaper;
    MoveL Offs(pOrigin,248.94,111.25,0.00),v40,z0,tPen\WObj:=wPaper;
    MoveL Offs(pOrigin,248.30,112.53,0.00),v40,z0,tPen\WObj:=wPaper;
    MoveL Offs(pOrigin,248.30,114.01,0.00),v40,z0,tPen\WObj:=wPaper;
    MoveL Offs(pOrigin,249.72,115.78,0.00),v40,z0,tPen\WObj:=wPaper;
    MoveL Offs(pOrigin,251.70,116.14,0.00),v40,z0,tPen\WObj:=wPaper;
    MoveL Offs(pOrigin,253.19,115.29,0.00),v40,z0,tPen\WObj:=wPaper;
    MoveL Offs(pOrigin,254.04,113.16,0.00),v40,z0,tPen\WObj:=wPaper;
    MoveL Offs(pOrigin,253.19,111.04,0.00),v40,z0,tPen\WObj:=wPaper;
    MoveL Offs(pOrigin,253.19,111.25,0.00),v40,z0,tPen\WObj:=wPaper;
    MoveL Offs(pOrigin,253.40,111.68,0.00),v40,z0,tPen\WObj:=wPaper;
    MoveL Offs(pOrigin,253.19,111.25,0.00),v40,z0,tPen\WObj:=wPaper;
    MoveL Offs(pOrigin,252.55,110.82,0.00),v40,z0,tPen\WObj:=wPaper;
  ENDPROC

